(* PLC project Untitled1, Eindhoven University of Technology (TU/e) CIF to Structured Text 0.0 *)
(* stored: creationDateTime 1970-01-01T01:00:00 *)

TYPE STATE : STRUCT
  curTime : LREAL;
  dvar_M_BoolToEventsDH AT %Q* : enum_E;
  dvar_M_BoolToEventsP AT %Q* : enum_E;
  dvar_M_BoolToEventsS AT %Q* : enum_E;
  dvar_M_BoolToEventsTB AT %Q* : enum_E;
  cvar_M_BTimer1_t AT %Q* : LREAL;
  dvar_M_BTimer1 AT %Q* : enum_E;
  dvar_M_HardwareMapDH_out_a_Dstartled AT %Q* : BOOL;
  dvar_M_HardwareMapDH_out_a_Dresetled AT %Q* : BOOL;
  dvar_M_HardwareMapDH_out_a_DledQ1 AT %Q* : BOOL;
  dvar_M_HardwareMapDH_out_a_DledQ2 AT %Q* : BOOL;
  dvar_M_HardwareMapDH_out_a_Dout4 AT %Q* : BOOL;
  dvar_M_HardwareMapDH_out_a_Dout5 AT %Q* : BOOL;
  dvar_M_HardwareMapDH_out_a_Dout6 AT %Q* : BOOL;
  dvar_M_HardwareMapDH_out_a_Dout7 AT %Q* : BOOL;
  dvar_M_HardwareMapDH_out_a_pusher1 AT %Q* : BOOL;
  dvar_M_HardwareMapDH_out_a_pusher2 AT %Q* : BOOL;
  dvar_M_HardwareMapDH_out_a_pusher3 AT %Q* : BOOL;
  dvar_M_HardwareMapDH_out_a_Hstartled AT %Q* : BOOL;
  dvar_M_HardwareMapDH_out_a_Hresetled AT %Q* : BOOL;
  dvar_M_HardwareMapDH_out_a_HledQ1 AT %Q* : BOOL;
  dvar_M_HardwareMapDH_out_a_HledQ2 AT %Q* : BOOL;
  dvar_M_HardwareMapDH_out_a_Hout4 AT %Q* : BOOL;
  dvar_M_HardwareMapDH_out_a_Hout5 AT %Q* : BOOL;
  dvar_M_HardwareMapDH_out_a_Hout6 AT %Q* : BOOL;
  dvar_M_HardwareMapDH_out_a_Hout7 AT %Q* : BOOL;
  dvar_M_HardwareMapDH_out_a_x2distributing AT %Q* : BOOL;
  dvar_M_HardwareMapDH_out_a_x2testing AT %Q* : BOOL;
  dvar_M_HardwareMapDH_out_a_zdown AT %Q* : BOOL;
  dvar_M_HardwareMapDH_out_a_gripperclose AT %Q* : BOOL;
  dvar_M_HardwareMapDH_out_a_transfer2pickpos AT %Q* : BOOL;
  dvar_M_HardwareMapDH_out_a_transfer2droppos AT %Q* : BOOL;
  dvar_M_HardwareMapDH_out_a_vacuum AT %Q* : BOOL;
  dvar_M_HardwareMapDH_out_a_ejectpulse AT %Q* : BOOL;
  dvar_M_HardwareMapDH_out_a_handlingready AT %Q* : BOOL;
  dvar_M_HardwareMapDH_init_err_sen_idx AT %Q* : DINT;
  dvar_M_HardwareMapDH_init_err_led_idx AT %Q* : DINT;
  cvar_M_HardwareMapDH_t AT %Q* : LREAL;
  dvar_M_HardwareMapDH AT %Q* : enum_E;
  dvar_M_HardwareMapP_out_a_Pstartled AT %Q* : BOOL;
  dvar_M_HardwareMapP_out_a_Presetled AT %Q* : BOOL;
  dvar_M_HardwareMapP_out_a_PledQ1 AT %Q* : BOOL;
  dvar_M_HardwareMapP_out_a_PledQ2 AT %Q* : BOOL;
  dvar_M_HardwareMapP_out_a_Pout4 AT %Q* : BOOL;
  dvar_M_HardwareMapP_out_a_Pout5 AT %Q* : BOOL;
  dvar_M_HardwareMapP_out_a_Pout6 AT %Q* : BOOL;
  dvar_M_HardwareMapP_out_a_Pout7 AT %Q* : BOOL;
  dvar_M_HardwareMapP_out_a_drill AT %Q* : BOOL;
  dvar_M_HardwareMapP_out_a_turntable AT %Q* : BOOL;
  dvar_M_HardwareMapP_out_a_drilldown AT %Q* : BOOL;
  dvar_M_HardwareMapP_out_a_drillup AT %Q* : BOOL;
  dvar_M_HardwareMapP_out_a_clamp AT %Q* : BOOL;
  dvar_M_HardwareMapP_out_a_tester AT %Q* : BOOL;
  dvar_M_HardwareMapP_out_a_eject AT %Q* : BOOL;
  dvar_M_HardwareMapP_out_a_processingready AT %Q* : BOOL;
  dvar_M_HardwareMapP_init_err_sen_idx AT %Q* : DINT;
  dvar_M_HardwareMapP_init_err_led_idx AT %Q* : DINT;
  cvar_M_HardwareMapP_t AT %Q* : LREAL;
  dvar_M_HardwareMapP AT %Q* : enum_E;
  dvar_M_HardwareMapS_out_a_Sstartled AT %Q* : BOOL;
  dvar_M_HardwareMapS_out_a_Sresetled AT %Q* : BOOL;
  dvar_M_HardwareMapS_out_a_SledQ1 AT %Q* : BOOL;
  dvar_M_HardwareMapS_out_a_SledQ2 AT %Q* : BOOL;
  dvar_M_HardwareMapS_out_a_Sout4 AT %Q* : BOOL;
  dvar_M_HardwareMapS_out_a_Sout5 AT %Q* : BOOL;
  dvar_M_HardwareMapS_out_a_Sout6 AT %Q* : BOOL;
  dvar_M_HardwareMapS_out_a_Sout7 AT %Q* : BOOL;
  dvar_M_HardwareMapS_out_a_conveyer AT %Q* : BOOL;
  dvar_M_HardwareMapS_out_a_gate1 AT %Q* : BOOL;
  dvar_M_HardwareMapS_out_a_gate2 AT %Q* : BOOL;
  dvar_M_HardwareMapS_out_a_stopperretract AT %Q* : BOOL;
  dvar_M_HardwareMapS_out_a_sortingready AT %Q* : BOOL;
  dvar_M_HardwareMapS_init_err_sen_idx AT %Q* : DINT;
  dvar_M_HardwareMapS_init_err_led_idx AT %Q* : DINT;
  cvar_M_HardwareMapS_t AT %Q* : LREAL;
  dvar_M_HardwareMapS AT %Q* : enum_E;
  dvar_M_HardwareMapTB_out_a_Tstartled AT %Q* : BOOL;
  dvar_M_HardwareMapTB_out_a_Tresetled AT %Q* : BOOL;
  dvar_M_HardwareMapTB_out_a_TledQ1 AT %Q* : BOOL;
  dvar_M_HardwareMapTB_out_a_TledQ2 AT %Q* : BOOL;
  dvar_M_HardwareMapTB_out_a_Tout4 AT %Q* : BOOL;
  dvar_M_HardwareMapTB_out_a_Tout5 AT %Q* : BOOL;
  dvar_M_HardwareMapTB_out_a_Tout6 AT %Q* : BOOL;
  dvar_M_HardwareMapTB_out_a_Tout7 AT %Q* : BOOL;
  dvar_M_HardwareMapTB_out_a_elevator_up AT %Q* : BOOL;
  dvar_M_HardwareMapTB_out_a_elevator_down AT %Q* : BOOL;
  dvar_M_HardwareMapTB_out_a_pusher AT %Q* : BOOL;
  dvar_M_HardwareMapTB_out_a_airslide AT %Q* : BOOL;
  dvar_M_HardwareMapTB_out_a_testingready AT %Q* : BOOL;
  dvar_M_HardwareMapTB_out_a_Bstartled AT %Q* : BOOL;
  dvar_M_HardwareMapTB_out_a_Bresetled AT %Q* : BOOL;
  dvar_M_HardwareMapTB_out_a_BledQ1 AT %Q* : BOOL;
  dvar_M_HardwareMapTB_out_a_BledQ2 AT %Q* : BOOL;
  dvar_M_HardwareMapTB_out_a_Bout4 AT %Q* : BOOL;
  dvar_M_HardwareMapTB_out_a_Bout5 AT %Q* : BOOL;
  dvar_M_HardwareMapTB_out_a_Bout6 AT %Q* : BOOL;
  dvar_M_HardwareMapTB_out_a_Bout7 AT %Q* : BOOL;
  dvar_M_HardwareMapTB_out_a_separator AT %Q* : BOOL;
  dvar_M_HardwareMapTB_out_a_conveyerB AT %Q* : BOOL;
  dvar_M_HardwareMapTB_out_a_bufferingready AT %Q* : BOOL;
  dvar_M_HardwareMapTB_init_err_sen_idx AT %Q* : DINT;
  dvar_M_HardwareMapTB_init_err_led_idx AT %Q* : DINT;
  cvar_M_HardwareMapTB_t AT %Q* : LREAL;
  dvar_M_HardwareMapTB AT %Q* : enum_E;
  cvar_M_STimer1_t AT %Q* : LREAL;
  dvar_M_STimer1 AT %Q* : enum_E;
  dvar_M_sup_A_airslide AT %Q* : enum_E;
  dvar_M_sup_A_bufferingready AT %Q* : enum_E;
  dvar_M_sup_A_clamp AT %Q* : enum_E;
  dvar_M_sup_A_conveyer AT %Q* : enum_E;
  dvar_M_sup_A_conveyerB AT %Q* : enum_E;
  dvar_M_sup_A_drill AT %Q* : enum_E;
  dvar_M_sup_A_drilldown AT %Q* : enum_E;
  dvar_M_sup_A_drillup AT %Q* : enum_E;
  dvar_M_sup_A_eject AT %Q* : enum_E;
  dvar_M_sup_A_ejectpulse AT %Q* : enum_E;
  dvar_M_sup_A_elevator_down AT %Q* : enum_E;
  dvar_M_sup_A_elevator_up AT %Q* : enum_E;
  dvar_M_sup_A_gate1 AT %Q* : enum_E;
  dvar_M_sup_A_gate2 AT %Q* : enum_E;
  dvar_M_sup_A_gripperclose AT %Q* : enum_E;
  dvar_M_sup_A_handlingready AT %Q* : enum_E;
  dvar_M_sup_A_processingready AT %Q* : enum_E;
  dvar_M_sup_A_pusher AT %Q* : enum_E;
  dvar_M_sup_A_pusher1 AT %Q* : enum_E;
  dvar_M_sup_A_pusher2 AT %Q* : enum_E;
  dvar_M_sup_A_pusher3 AT %Q* : enum_E;
  dvar_M_sup_A_separator AT %Q* : enum_E;
  dvar_M_sup_A_sortingready AT %Q* : enum_E;
  dvar_M_sup_A_stopperretract AT %Q* : enum_E;
  dvar_M_sup_A_tester AT %Q* : enum_E;
  dvar_M_sup_A_testingready AT %Q* : enum_E;
  dvar_M_sup_A_transfer2droppos AT %Q* : enum_E;
  dvar_M_sup_A_transfer2pickpos AT %Q* : enum_E;
  dvar_M_sup_A_turntable AT %Q* : enum_E;
  dvar_M_sup_A_vacuum AT %Q* : enum_E;
  dvar_M_sup_A_x2distributing AT %Q* : enum_E;
  dvar_M_sup_A_x2testing AT %Q* : enum_E;
  dvar_M_sup_A_zdown AT %Q* : enum_E;
  dvar_M_sup_BDynamics AT %Q* : enum_E;
  dvar_M_sup_BTimer AT %Q* : enum_E;
  dvar_M_sup_ClampDrill AT %Q* : enum_E;
  dvar_M_sup_DDynamics1 AT %Q* : enum_E;
  dvar_M_sup_DDynamics2 AT %Q* : enum_E;
  dvar_M_sup_DDynamics3 AT %Q* : enum_E;
  dvar_M_sup_HDynamics1 AT %Q* : enum_E;
  dvar_M_sup_HDynamics2 AT %Q* : enum_E;
  dvar_M_sup_HDynamics3 AT %Q* : enum_E;
  dvar_M_sup_PDynamics AT %Q* : enum_E;
  dvar_M_sup_PusherLift AT %Q* : enum_E;
  dvar_M_sup_S_atdrill AT %Q* : enum_E;
  dvar_M_sup_S_atend AT %Q* : enum_E;
  dvar_M_sup_S_atexit AT %Q* : enum_E;
  dvar_M_sup_S_atin AT %Q* : enum_E;
  dvar_M_sup_S_atinput AT %Q* : enum_E;
  dvar_M_sup_S_atseparator AT %Q* : enum_E;
  dvar_M_sup_S_atspare AT %Q* : enum_E;
  dvar_M_sup_S_attest AT %Q* : enum_E;
  dvar_M_sup_S_Binitialized AT %Q* : enum_E;
  dvar_M_sup_S_bufferingbusy AT %Q* : enum_E;
  dvar_M_sup_S_capacitive AT %Q* : enum_E;
  dvar_M_sup_S_clamp AT %Q* : enum_E;
  dvar_M_sup_S_Dinitialized AT %Q* : enum_E;
  dvar_M_sup_S_drill_down AT %Q* : enum_E;
  dvar_M_sup_S_drill_up AT %Q* : enum_E;
  dvar_M_sup_S_elevator_down AT %Q* : enum_E;
  dvar_M_sup_S_elevator_up AT %Q* : enum_E;
  dvar_M_sup_S_gate1_closed AT %Q* : enum_E;
  dvar_M_sup_S_gate1_opened AT %Q* : enum_E;
  dvar_M_sup_S_gate2_closed AT %Q* : enum_E;
  dvar_M_sup_S_gate2_opened AT %Q* : enum_E;
  dvar_M_sup_S_gripper AT %Q* : enum_E;
  dvar_M_sup_S_handlingbusy AT %Q* : enum_E;
  dvar_M_sup_S_Hinitialized AT %Q* : enum_E;
  dvar_M_sup_S_inductive AT %Q* : enum_E;
  dvar_M_sup_S_optical AT %Q* : enum_E;
  dvar_M_sup_S_opticalT AT %Q* : enum_E;
  dvar_M_sup_S_Pinitialized AT %Q* : enum_E;
  dvar_M_sup_S_processingbusy AT %Q* : enum_E;
  dvar_M_sup_S_product AT %Q* : enum_E;
  dvar_M_sup_S_product1 AT %Q* : enum_E;
  dvar_M_sup_S_product2 AT %Q* : enum_E;
  dvar_M_sup_S_product3 AT %Q* : enum_E;
  dvar_M_sup_S_product4 AT %Q* : enum_E;
  dvar_M_sup_S_productheight AT %Q* : enum_E;
  dvar_M_sup_S_pusher AT %Q* : enum_E;
  dvar_M_sup_S_pusher1_in AT %Q* : enum_E;
  dvar_M_sup_S_pusher1_out AT %Q* : enum_E;
  dvar_M_sup_S_pusher2_in AT %Q* : enum_E;
  dvar_M_sup_S_pusher2_out AT %Q* : enum_E;
  dvar_M_sup_S_pusher3_in AT %Q* : enum_E;
  dvar_M_sup_S_pusher3_out AT %Q* : enum_E;
  dvar_M_sup_S_reflective AT %Q* : enum_E;
  dvar_M_sup_S_separator_closed AT %Q* : enum_E;
  dvar_M_sup_S_separator_opened AT %Q* : enum_E;
  dvar_M_sup_S_Sinitialized AT %Q* : enum_E;
  dvar_M_sup_S_slidefull AT %Q* : enum_E;
  dvar_M_sup_S_sortingbusy AT %Q* : enum_E;
  dvar_M_sup_S_stack1_filled AT %Q* : enum_E;
  dvar_M_sup_S_stack2_filled AT %Q* : enum_E;
  dvar_M_sup_S_stack3_filled AT %Q* : enum_E;
  dvar_M_sup_S_test_ok AT %Q* : enum_E;
  dvar_M_sup_S_testingbusy AT %Q* : enum_E;
  dvar_M_sup_S_Tinitialized AT %Q* : enum_E;
  dvar_M_sup_S_transfer_atdrop AT %Q* : enum_E;
  dvar_M_sup_S_transfer_athalfway AT %Q* : enum_E;
  dvar_M_sup_S_transfer_atpickup AT %Q* : enum_E;
  dvar_M_sup_S_turntable AT %Q* : enum_E;
  dvar_M_sup_S_vacuum AT %Q* : enum_E;
  dvar_M_sup_S_xpos_at1 AT %Q* : enum_E;
  dvar_M_sup_S_xpos_at2 AT %Q* : enum_E;
  dvar_M_sup_S_xpos_at3 AT %Q* : enum_E;
  dvar_M_sup_S_xpos_atdrop AT %Q* : enum_E;
  dvar_M_sup_S_zpos_atdown AT %Q* : enum_E;
  dvar_M_sup_S_zpos_atup AT %Q* : enum_E;
  dvar_M_sup_SDynamics1 AT %Q* : enum_E;
  dvar_M_sup_SDynamics2 AT %Q* : enum_E;
  dvar_M_sup_STimer AT %Q* : enum_E;
  dvar_M_sup_sup AT %Q* : enum_E;
  dvar_M_sup_TDynamics AT %Q* : enum_E;
  dvar_M_sup_Tester AT %Q* : enum_E;
  dvar_M_sup_Timer AT %Q* : enum_E;
  dvar_M_sup_TTimer AT %Q* : enum_E;
  cvar_M_Timer1_t AT %Q* : LREAL;
  dvar_M_Timer1 AT %Q* : enum_E;
  cvar_M_TTimer1_t AT %Q* : LREAL;
  dvar_M_TTimer1 AT %Q* : enum_E;
END_STRUCT;
END_TYPE

TYPE enum_E : (elit_eight, elit_five, elit_Four, elit_four2, elit_init0, elit_init1, elit_init2, elit_init3, elit_init4, elit_init5, elit_init6, elit_init7, elit_init8, elit_init9, elit_init_error, elit_init_ok, elit_init_sensor_check, elit_initialized, elit_nine, elit_Off, elit_On, elit_One, elit_one2, elit_Running, elit_seven, elit_six, elit_Three, elit_three2, elit_Timeout, elit_Two, elit_two2, elit_X);
END_TYPE

FUNCTION ifExprFunc1 : LREAL
  VAR_INPUT
    state : STATE;
  END_VAR

            IF ((state.dvar_M_BTimer1) = (elit_Running)) THEN
    ifExprFunc1 := 1.0;
ELSE
    ifExprFunc1 := 0.0;
END_IF;
          
END_FUNCTION

FUNCTION derivcvar_M_BTimer1_t : LREAL
  VAR_INPUT
    state : STATE;
  END_VAR

            derivcvar_M_BTimer1_t := ifExprFunc1(state);
          
END_FUNCTION

FUNCTION derivcvar_M_HardwareMapDH_t : LREAL
  VAR_INPUT
    state : STATE;
  END_VAR

            derivcvar_M_HardwareMapDH_t := 1.0;
          
END_FUNCTION

FUNCTION derivcvar_M_HardwareMapP_t : LREAL
  VAR_INPUT
    state : STATE;
  END_VAR

            derivcvar_M_HardwareMapP_t := 1.0;
          
END_FUNCTION

FUNCTION derivcvar_M_HardwareMapS_t : LREAL
  VAR_INPUT
    state : STATE;
  END_VAR

            derivcvar_M_HardwareMapS_t := 1.0;
          
END_FUNCTION

FUNCTION derivcvar_M_HardwareMapTB_t : LREAL
  VAR_INPUT
    state : STATE;
  END_VAR

            derivcvar_M_HardwareMapTB_t := 1.0;
          
END_FUNCTION

FUNCTION ifExprFunc2 : LREAL
  VAR_INPUT
    state : STATE;
  END_VAR

            IF ((state.dvar_M_STimer1) = (elit_Running)) THEN
    ifExprFunc2 := 1.0;
ELSE
    ifExprFunc2 := 0.0;
END_IF;
          
END_FUNCTION

FUNCTION derivcvar_M_STimer1_t : LREAL
  VAR_INPUT
    state : STATE;
  END_VAR

            derivcvar_M_STimer1_t := ifExprFunc2(state);
          
END_FUNCTION

FUNCTION ifExprFunc3 : LREAL
  VAR_INPUT
    state : STATE;
  END_VAR

            IF ((state.dvar_M_Timer1) = (elit_Running)) THEN
    ifExprFunc3 := 1.0;
ELSE
    ifExprFunc3 := 0.0;
END_IF;
          
END_FUNCTION

FUNCTION derivcvar_M_Timer1_t : LREAL
  VAR_INPUT
    state : STATE;
  END_VAR

            derivcvar_M_Timer1_t := ifExprFunc3(state);
          
END_FUNCTION

FUNCTION ifExprFunc4 : LREAL
  VAR_INPUT
    state : STATE;
  END_VAR

            IF ((state.dvar_M_TTimer1) = (elit_Running)) THEN
    ifExprFunc4 := 1.0;
ELSE
    ifExprFunc4 := 0.0;
END_IF;
          
END_FUNCTION

FUNCTION derivcvar_M_TTimer1_t : LREAL
  VAR_INPUT
    state : STATE;
  END_VAR

            derivcvar_M_TTimer1_t := ifExprFunc4(state);
          
END_FUNCTION

PROGRAM MAIN
  VAR_OUTPUT
    timerValue0 : TIME;
    timerValue1 : TIME;
  END_VAR
  VAR
    cnt : LINT;
    first : BOOL := TRUE;
    curTimerValue : TIME;
    state0 : STATE;
    curTime : LREAL;
    loopsKilled : LINT;
  END_VAR
  VAR_TEMP
    lastTimerValue : TIME;
    curDeltaTime : TIME;
    curDeltaSecs : LREAL;
    state1 : STATE;
    progress : BOOL;
    loopCount : INT;
    b1 : BOOL;
    b2 : BOOL;
    b3 : BOOL;
    b4 : BOOL;
  END_VAR

            
// Handle 'time' and cycle time.
cnt := cnt + 1;

timer0(IN := curTimer = 0, PT := T#1D);
timer1(IN := curTimer = 1, PT := T#1D);
timerValue0 := timer0.ET;
timerValue1 := timer1.ET;

lastTimerValue := curTimerValue;
IF curTimer = 0 THEN
    curTimerValue := timerValue0;
ELSE
    curTimerValue := timerValue1;
END_IF;
curDeltaTime := curTimerValue - lastTimerValue;
curDeltaSecs := TIME_TO_LREAL(curDeltaTime) / 1000;
curTime := curTime + curDeltaSecs;

IF cnt MOD 10 = 0 THEN
    curTimer := 1 - curTimer;
    curTimerValue := T#0S;
    timer0(IN := curTimer = 0, PT := T#1D);
    timer1(IN := curTimer = 1, PT := T#1D);
    timerValue0 := timer0.ET;
    timerValue1 := timer1.ET;
END_IF;

IF first THEN
    first := FALSE;

    // Initialize state variables for initial state.
    state0.dvar_M_BoolToEventsDH := elit_X;
    state0.dvar_M_BoolToEventsP := elit_X;
    state0.dvar_M_BoolToEventsS := elit_X;
    state0.dvar_M_BoolToEventsTB := elit_X;
    state0.cvar_M_BTimer1_t := 0.0;
    state0.dvar_M_BTimer1 := elit_Off;
    state0.dvar_M_HardwareMapDH_out_a_Dstartled := FALSE;
    state0.dvar_M_HardwareMapDH_out_a_Dresetled := FALSE;
    state0.dvar_M_HardwareMapDH_out_a_DledQ1 := TRUE;
    state0.dvar_M_HardwareMapDH_out_a_DledQ2 := TRUE;
    state0.dvar_M_HardwareMapDH_out_a_Dout4 := FALSE;
    state0.dvar_M_HardwareMapDH_out_a_Dout5 := FALSE;
    state0.dvar_M_HardwareMapDH_out_a_Dout6 := FALSE;
    state0.dvar_M_HardwareMapDH_out_a_Dout7 := FALSE;
    state0.dvar_M_HardwareMapDH_out_a_pusher1 := FALSE;
    state0.dvar_M_HardwareMapDH_out_a_pusher2 := FALSE;
    state0.dvar_M_HardwareMapDH_out_a_pusher3 := FALSE;
    state0.dvar_M_HardwareMapDH_out_a_Hstartled := FALSE;
    state0.dvar_M_HardwareMapDH_out_a_Hresetled := FALSE;
    state0.dvar_M_HardwareMapDH_out_a_HledQ1 := TRUE;
    state0.dvar_M_HardwareMapDH_out_a_HledQ2 := TRUE;
    state0.dvar_M_HardwareMapDH_out_a_Hout4 := FALSE;
    state0.dvar_M_HardwareMapDH_out_a_Hout5 := FALSE;
    state0.dvar_M_HardwareMapDH_out_a_Hout6 := FALSE;
    state0.dvar_M_HardwareMapDH_out_a_Hout7 := FALSE;
    state0.dvar_M_HardwareMapDH_out_a_x2distributing := TRUE;
    state0.dvar_M_HardwareMapDH_out_a_x2testing := TRUE;
    state0.dvar_M_HardwareMapDH_out_a_zdown := FALSE;
    state0.dvar_M_HardwareMapDH_out_a_gripperclose := FALSE;
    state0.dvar_M_HardwareMapDH_out_a_transfer2pickpos := FALSE;
    state0.dvar_M_HardwareMapDH_out_a_transfer2droppos := FALSE;
    state0.dvar_M_HardwareMapDH_out_a_vacuum := FALSE;
    state0.dvar_M_HardwareMapDH_out_a_ejectpulse := FALSE;
    state0.dvar_M_HardwareMapDH_out_a_handlingready := FALSE;
    state0.dvar_M_HardwareMapDH_init_err_sen_idx := -1;
    state0.dvar_M_HardwareMapDH_init_err_led_idx := 0;
    state0.cvar_M_HardwareMapDH_t := 0.0;
    state0.dvar_M_HardwareMapDH := elit_init0;
    state0.dvar_M_HardwareMapP_out_a_Pstartled := FALSE;
    state0.dvar_M_HardwareMapP_out_a_Presetled := FALSE;
    state0.dvar_M_HardwareMapP_out_a_PledQ1 := TRUE;
    state0.dvar_M_HardwareMapP_out_a_PledQ2 := TRUE;
    state0.dvar_M_HardwareMapP_out_a_Pout4 := FALSE;
    state0.dvar_M_HardwareMapP_out_a_Pout5 := FALSE;
    state0.dvar_M_HardwareMapP_out_a_Pout6 := FALSE;
    state0.dvar_M_HardwareMapP_out_a_Pout7 := FALSE;
    state0.dvar_M_HardwareMapP_out_a_drill := FALSE;
    state0.dvar_M_HardwareMapP_out_a_turntable := FALSE;
    state0.dvar_M_HardwareMapP_out_a_drilldown := FALSE;
    state0.dvar_M_HardwareMapP_out_a_drillup := TRUE;
    state0.dvar_M_HardwareMapP_out_a_clamp := FALSE;
    state0.dvar_M_HardwareMapP_out_a_tester := FALSE;
    state0.dvar_M_HardwareMapP_out_a_eject := FALSE;
    state0.dvar_M_HardwareMapP_out_a_processingready := FALSE;
    state0.dvar_M_HardwareMapP_init_err_sen_idx := -1;
    state0.dvar_M_HardwareMapP_init_err_led_idx := 0;
    state0.cvar_M_HardwareMapP_t := 0.0;
    state0.dvar_M_HardwareMapP := elit_init0;
    state0.dvar_M_HardwareMapS_out_a_Sstartled := FALSE;
    state0.dvar_M_HardwareMapS_out_a_Sresetled := FALSE;
    state0.dvar_M_HardwareMapS_out_a_SledQ1 := TRUE;
    state0.dvar_M_HardwareMapS_out_a_SledQ2 := TRUE;
    state0.dvar_M_HardwareMapS_out_a_Sout4 := FALSE;
    state0.dvar_M_HardwareMapS_out_a_Sout5 := FALSE;
    state0.dvar_M_HardwareMapS_out_a_Sout6 := FALSE;
    state0.dvar_M_HardwareMapS_out_a_Sout7 := FALSE;
    state0.dvar_M_HardwareMapS_out_a_conveyer := FALSE;
    state0.dvar_M_HardwareMapS_out_a_gate1 := FALSE;
    state0.dvar_M_HardwareMapS_out_a_gate2 := FALSE;
    state0.dvar_M_HardwareMapS_out_a_stopperretract := FALSE;
    state0.dvar_M_HardwareMapS_out_a_sortingready := FALSE;
    state0.dvar_M_HardwareMapS_init_err_sen_idx := -1;
    state0.dvar_M_HardwareMapS_init_err_led_idx := 0;
    state0.cvar_M_HardwareMapS_t := 0.0;
    state0.dvar_M_HardwareMapS := elit_init0;
    state0.dvar_M_HardwareMapTB_out_a_Tstartled := FALSE;
    state0.dvar_M_HardwareMapTB_out_a_Tresetled := FALSE;
    state0.dvar_M_HardwareMapTB_out_a_TledQ1 := TRUE;
    state0.dvar_M_HardwareMapTB_out_a_TledQ2 := TRUE;
    state0.dvar_M_HardwareMapTB_out_a_Tout4 := FALSE;
    state0.dvar_M_HardwareMapTB_out_a_Tout5 := FALSE;
    state0.dvar_M_HardwareMapTB_out_a_Tout6 := FALSE;
    state0.dvar_M_HardwareMapTB_out_a_Tout7 := FALSE;
    state0.dvar_M_HardwareMapTB_out_a_elevator_up := FALSE;
    state0.dvar_M_HardwareMapTB_out_a_elevator_down := TRUE;
    state0.dvar_M_HardwareMapTB_out_a_pusher := FALSE;
    state0.dvar_M_HardwareMapTB_out_a_airslide := FALSE;
    state0.dvar_M_HardwareMapTB_out_a_testingready := FALSE;
    state0.dvar_M_HardwareMapTB_out_a_Bstartled := FALSE;
    state0.dvar_M_HardwareMapTB_out_a_Bresetled := FALSE;
    state0.dvar_M_HardwareMapTB_out_a_BledQ1 := TRUE;
    state0.dvar_M_HardwareMapTB_out_a_BledQ2 := TRUE;
    state0.dvar_M_HardwareMapTB_out_a_Bout4 := FALSE;
    state0.dvar_M_HardwareMapTB_out_a_Bout5 := FALSE;
    state0.dvar_M_HardwareMapTB_out_a_Bout6 := FALSE;
    state0.dvar_M_HardwareMapTB_out_a_Bout7 := FALSE;
    state0.dvar_M_HardwareMapTB_out_a_separator := FALSE;
    state0.dvar_M_HardwareMapTB_out_a_conveyerB := FALSE;
    state0.dvar_M_HardwareMapTB_out_a_bufferingready := FALSE;
    state0.dvar_M_HardwareMapTB_init_err_sen_idx := -1;
    state0.dvar_M_HardwareMapTB_init_err_led_idx := 0;
    state0.cvar_M_HardwareMapTB_t := 0.0;
    state0.dvar_M_HardwareMapTB := elit_init0;
    state0.cvar_M_STimer1_t := 0.0;
    state0.dvar_M_STimer1 := elit_Off;
    state0.dvar_M_sup_A_airslide := elit_Off;
    state0.dvar_M_sup_A_bufferingready := elit_Off;
    state0.dvar_M_sup_A_clamp := elit_Off;
    state0.dvar_M_sup_A_conveyer := elit_Off;
    state0.dvar_M_sup_A_conveyerB := elit_Off;
    state0.dvar_M_sup_A_drill := elit_Off;
    state0.dvar_M_sup_A_drilldown := elit_Off;
    state0.dvar_M_sup_A_drillup := elit_On;
    state0.dvar_M_sup_A_eject := elit_Off;
    state0.dvar_M_sup_A_ejectpulse := elit_Off;
    state0.dvar_M_sup_A_elevator_down := elit_On;
    state0.dvar_M_sup_A_elevator_up := elit_Off;
    state0.dvar_M_sup_A_gate1 := elit_Off;
    state0.dvar_M_sup_A_gate2 := elit_Off;
    state0.dvar_M_sup_A_gripperclose := elit_Off;
    state0.dvar_M_sup_A_handlingready := elit_Off;
    state0.dvar_M_sup_A_processingready := elit_Off;
    state0.dvar_M_sup_A_pusher := elit_Off;
    state0.dvar_M_sup_A_pusher1 := elit_Off;
    state0.dvar_M_sup_A_pusher2 := elit_Off;
    state0.dvar_M_sup_A_pusher3 := elit_Off;
    state0.dvar_M_sup_A_separator := elit_On;
    state0.dvar_M_sup_A_sortingready := elit_Off;
    state0.dvar_M_sup_A_stopperretract := elit_Off;
    state0.dvar_M_sup_A_tester := elit_Off;
    state0.dvar_M_sup_A_testingready := elit_Off;
    state0.dvar_M_sup_A_transfer2droppos := elit_Off;
    state0.dvar_M_sup_A_transfer2pickpos := elit_Off;
    state0.dvar_M_sup_A_turntable := elit_Off;
    state0.dvar_M_sup_A_vacuum := elit_Off;
    state0.dvar_M_sup_A_x2distributing := elit_On;
    state0.dvar_M_sup_A_x2testing := elit_On;
    state0.dvar_M_sup_A_zdown := elit_Off;
    state0.dvar_M_sup_BDynamics := elit_X;
    state0.dvar_M_sup_BTimer := elit_Off;
    state0.dvar_M_sup_ClampDrill := elit_one2;
    state0.dvar_M_sup_DDynamics1 := elit_X;
    state0.dvar_M_sup_DDynamics2 := elit_X;
    state0.dvar_M_sup_DDynamics3 := elit_X;
    state0.dvar_M_sup_HDynamics1 := elit_X;
    state0.dvar_M_sup_HDynamics2 := elit_X;
    state0.dvar_M_sup_HDynamics3 := elit_X;
    state0.dvar_M_sup_PDynamics := elit_X;
    state0.dvar_M_sup_PusherLift := elit_One;
    state0.dvar_M_sup_S_atdrill := elit_Off;
    state0.dvar_M_sup_S_atend := elit_Off;
    state0.dvar_M_sup_S_atexit := elit_Off;
    state0.dvar_M_sup_S_atin := elit_Off;
    state0.dvar_M_sup_S_atinput := elit_Off;
    state0.dvar_M_sup_S_atseparator := elit_Off;
    state0.dvar_M_sup_S_atspare := elit_Off;
    state0.dvar_M_sup_S_attest := elit_Off;
    state0.dvar_M_sup_S_Binitialized := elit_Off;
    state0.dvar_M_sup_S_bufferingbusy := elit_On;
    state0.dvar_M_sup_S_capacitive := elit_Off;
    state0.dvar_M_sup_S_clamp := elit_Off;
    state0.dvar_M_sup_S_Dinitialized := elit_Off;
    state0.dvar_M_sup_S_drill_down := elit_Off;
    state0.dvar_M_sup_S_drill_up := elit_On;
    state0.dvar_M_sup_S_elevator_down := elit_On;
    state0.dvar_M_sup_S_elevator_up := elit_Off;
    state0.dvar_M_sup_S_gate1_closed := elit_Off;
    state0.dvar_M_sup_S_gate1_opened := elit_On;
    state0.dvar_M_sup_S_gate2_closed := elit_Off;
    state0.dvar_M_sup_S_gate2_opened := elit_On;
    state0.dvar_M_sup_S_gripper := elit_Off;
    state0.dvar_M_sup_S_handlingbusy := elit_On;
    state0.dvar_M_sup_S_Hinitialized := elit_Off;
    state0.dvar_M_sup_S_inductive := elit_Off;
    state0.dvar_M_sup_S_optical := elit_Off;
    state0.dvar_M_sup_S_opticalT := elit_Off;
    state0.dvar_M_sup_S_Pinitialized := elit_Off;
    state0.dvar_M_sup_S_processingbusy := elit_On;
    state0.dvar_M_sup_S_product := elit_Off;
    state0.dvar_M_sup_S_product1 := elit_Off;
    state0.dvar_M_sup_S_product2 := elit_Off;
    state0.dvar_M_sup_S_product3 := elit_Off;
    state0.dvar_M_sup_S_product4 := elit_Off;
    state0.dvar_M_sup_S_productheight := elit_Off;
    state0.dvar_M_sup_S_pusher := elit_Off;
    state0.dvar_M_sup_S_pusher1_in := elit_On;
    state0.dvar_M_sup_S_pusher1_out := elit_Off;
    state0.dvar_M_sup_S_pusher2_in := elit_On;
    state0.dvar_M_sup_S_pusher2_out := elit_Off;
    state0.dvar_M_sup_S_pusher3_in := elit_On;
    state0.dvar_M_sup_S_pusher3_out := elit_Off;
    state0.dvar_M_sup_S_reflective := elit_Off;
    state0.dvar_M_sup_S_separator_closed := elit_On;
    state0.dvar_M_sup_S_separator_opened := elit_Off;
    state0.dvar_M_sup_S_Sinitialized := elit_Off;
    state0.dvar_M_sup_S_slidefull := elit_Off;
    state0.dvar_M_sup_S_sortingbusy := elit_On;
    state0.dvar_M_sup_S_stack1_filled := elit_On;
    state0.dvar_M_sup_S_stack2_filled := elit_On;
    state0.dvar_M_sup_S_stack3_filled := elit_On;
    state0.dvar_M_sup_S_test_ok := elit_Off;
    state0.dvar_M_sup_S_testingbusy := elit_On;
    state0.dvar_M_sup_S_Tinitialized := elit_Off;
    state0.dvar_M_sup_S_transfer_atdrop := elit_Off;
    state0.dvar_M_sup_S_transfer_athalfway := elit_On;
    state0.dvar_M_sup_S_transfer_atpickup := elit_Off;
    state0.dvar_M_sup_S_turntable := elit_On;
    state0.dvar_M_sup_S_vacuum := elit_Off;
    state0.dvar_M_sup_S_xpos_at1 := elit_Off;
    state0.dvar_M_sup_S_xpos_at2 := elit_Off;
    state0.dvar_M_sup_S_xpos_at3 := elit_Off;
    state0.dvar_M_sup_S_xpos_atdrop := elit_On;
    state0.dvar_M_sup_S_zpos_atdown := elit_Off;
    state0.dvar_M_sup_S_zpos_atup := elit_On;
    state0.dvar_M_sup_SDynamics1 := elit_X;
    state0.dvar_M_sup_SDynamics2 := elit_X;
    state0.dvar_M_sup_STimer := elit_Off;
    state0.dvar_M_sup_sup := elit_X;
    state0.dvar_M_sup_TDynamics := elit_X;
    state0.dvar_M_sup_Tester := elit_One;
    state0.dvar_M_sup_Timer := elit_Off;
    state0.dvar_M_sup_TTimer := elit_Off;
    state0.cvar_M_Timer1_t := 0.0;
    state0.dvar_M_Timer1 := elit_Off;
    state0.cvar_M_TTimer1_t := 0.0;
    state0.dvar_M_TTimer1 := elit_Off;
ELSE
    // Update continuous variables for time delay.
    state1.cvar_M_BTimer1_t := state0.cvar_M_BTimer1_t + curDeltaSecs * derivcvar_M_BTimer1_t(state0);
    state1.cvar_M_HardwareMapDH_t := state0.cvar_M_HardwareMapDH_t + curDeltaSecs * derivcvar_M_HardwareMapDH_t(state0);
    state1.cvar_M_HardwareMapP_t := state0.cvar_M_HardwareMapP_t + curDeltaSecs * derivcvar_M_HardwareMapP_t(state0);
    state1.cvar_M_HardwareMapS_t := state0.cvar_M_HardwareMapS_t + curDeltaSecs * derivcvar_M_HardwareMapS_t(state0);
    state1.cvar_M_HardwareMapTB_t := state0.cvar_M_HardwareMapTB_t + curDeltaSecs * derivcvar_M_HardwareMapTB_t(state0);
    state1.cvar_M_STimer1_t := state0.cvar_M_STimer1_t + curDeltaSecs * derivcvar_M_STimer1_t(state0);
    state1.cvar_M_Timer1_t := state0.cvar_M_Timer1_t + curDeltaSecs * derivcvar_M_Timer1_t(state0);
    state1.cvar_M_TTimer1_t := state0.cvar_M_TTimer1_t + curDeltaSecs * derivcvar_M_TTimer1_t(state0);

    state0.curTime := curTime;
    state0.cvar_M_BTimer1_t := state1.cvar_M_BTimer1_t;
    state0.cvar_M_HardwareMapDH_t := state1.cvar_M_HardwareMapDH_t;
    state0.cvar_M_HardwareMapP_t := state1.cvar_M_HardwareMapP_t;
    state0.cvar_M_HardwareMapS_t := state1.cvar_M_HardwareMapS_t;
    state0.cvar_M_HardwareMapTB_t := state1.cvar_M_HardwareMapTB_t;
    state0.cvar_M_STimer1_t := state1.cvar_M_STimer1_t;
    state0.cvar_M_Timer1_t := state1.cvar_M_Timer1_t;
    state0.cvar_M_TTimer1_t := state1.cvar_M_TTimer1_t;
END_IF;

// Event loop.
WHILE TRUE DO
    progress := FALSE;

    // Event "A_airslide_c_off".
    IF NOT progress THEN
        b1 := (state0.dvar_M_sup_A_airslide) = (elit_On);
        b1 := b1 AND ((state0.dvar_M_sup_sup) = (elit_X));
        b1 := b1 AND ((state0.dvar_M_sup_S_elevator_down) = (elit_On));
        b1 := b1 AND ((state0.dvar_M_sup_S_Tinitialized) = (elit_On));
        IF b1 THEN
            progress := TRUE;
            state1 := state0;

            state1.dvar_M_sup_A_airslide := elit_Off;

            state0 := state1;
        END_IF;
    END_IF;

    // Event "A_airslide_c_on".
    IF NOT progress THEN
        b1 := (state0.dvar_M_sup_A_airslide) = (elit_Off);
        b1 := b1 AND ((state0.dvar_M_sup_sup) = (elit_X));
        b1 := b1 AND ((state0.dvar_M_sup_S_pusher) = (elit_On));
        b1 := b1 AND ((state0.dvar_M_sup_S_elevator_up) = (elit_On));
        b1 := b1 AND ((state0.dvar_M_sup_S_Tinitialized) = (elit_On));
        IF b1 THEN
            progress := TRUE;
            state1 := state0;

            state1.dvar_M_sup_A_airslide := elit_On;

            state0 := state1;
        END_IF;
    END_IF;

    // Event "A_bufferingready_c_off".
    IF NOT progress THEN
        b1 := (state0.dvar_M_sup_A_bufferingready) = (elit_On);
        b1 := b1 AND ((state0.dvar_M_sup_sup) = (elit_X));
        b1 := b1 AND ((state0.dvar_M_sup_S_Binitialized) = (elit_On));
        IF b1 THEN
            progress := TRUE;
            state1 := state0;

            state1.dvar_M_sup_A_bufferingready := elit_Off;

            state0 := state1;
        END_IF;
    END_IF;

    // Event "A_bufferingready_c_on".
    IF NOT progress THEN
        IF FALSE THEN
            progress := TRUE;
            state1 := state0;

            state1.dvar_M_sup_A_bufferingready := elit_On;

            state0 := state1;
        END_IF;
    END_IF;

    // Event "A_clamp_c_off".
    IF NOT progress THEN
        b1 := (state0.dvar_M_sup_A_clamp) = (elit_On);
        b1 := b1 AND ((state0.dvar_M_sup_ClampDrill) = (elit_eight));
        b1 := b1 AND ((state0.dvar_M_sup_sup) = (elit_X));
        b1 := b1 AND ((state0.dvar_M_sup_S_drill_up) = (elit_On));
        b1 := b1 AND ((state0.dvar_M_sup_S_Pinitialized) = (elit_On));
        IF b1 THEN
            progress := TRUE;
            state1 := state0;

            state1.dvar_M_sup_A_clamp := elit_Off;
            state1.dvar_M_sup_ClampDrill := elit_nine;

            state0 := state1;
        END_IF;
    END_IF;

    // Event "A_clamp_c_on".
    IF NOT progress THEN
        b1 := (state0.dvar_M_sup_A_clamp) = (elit_Off);
        b1 := b1 AND ((state0.dvar_M_sup_ClampDrill) = (elit_one2));
        b1 := b1 AND ((state0.dvar_M_sup_sup) = (elit_X));
        b1 := b1 AND ((state0.dvar_M_sup_A_turntable) = (elit_Off));
        b1 := b1 AND ((state0.dvar_M_sup_S_atdrill) = (elit_On));
        b1 := b1 AND ((state0.dvar_M_sup_S_Pinitialized) = (elit_On));
        b1 := b1 AND ((state0.dvar_M_sup_S_turntable) = (elit_On));
        b1 := b1 AND ((state0.dvar_M_sup_Timer) = (elit_Timeout));
        IF b1 THEN
            progress := TRUE;
            state1 := state0;

            state1.dvar_M_sup_A_clamp := elit_On;
            state1.dvar_M_sup_ClampDrill := elit_two2;

            state0 := state1;
        END_IF;
    END_IF;

    // Event "A_conveyer_c_off".
    IF NOT progress THEN
        b1 := (state0.dvar_M_sup_A_conveyer) = (elit_On);
        b1 := b1 AND ((state0.dvar_M_sup_sup) = (elit_X));
        b1 := b1 AND ((state0.dvar_M_sup_S_Sinitialized) = (elit_On));
        b1 := b1 AND ((state0.dvar_M_sup_S_slidefull) = (elit_On));
        IF b1 THEN
            progress := TRUE;
            state1 := state0;

            state1.dvar_M_sup_A_conveyer := elit_Off;

            state0 := state1;
        END_IF;
    END_IF;

    // Event "A_conveyer_c_on".
    IF NOT progress THEN
        b1 := (state0.dvar_M_sup_A_conveyer) = (elit_Off);
        b1 := b1 AND ((state0.dvar_M_sup_sup) = (elit_X));
        b1 := b1 AND ((state0.dvar_M_sup_S_product) = (elit_On));
        b1 := b1 AND ((state0.dvar_M_sup_S_Sinitialized) = (elit_On));
        IF b1 THEN
            progress := TRUE;
            state1 := state0;

            state1.dvar_M_sup_A_conveyer := elit_On;

            state0 := state1;
        END_IF;
    END_IF;

    // Event "A_conveyerB_c_off".
    IF NOT progress THEN
        b1 := (state0.dvar_M_sup_A_conveyerB) = (elit_On);
        b1 := b1 AND ((state0.dvar_M_sup_sup) = (elit_X));
        b1 := b1 AND ((state0.dvar_M_sup_BTimer) = (elit_Timeout));
        b1 := b1 AND ((state0.dvar_M_sup_S_Binitialized) = (elit_On));
        IF b1 THEN
            progress := TRUE;
            state1 := state0;

            state1.dvar_M_sup_A_conveyerB := elit_Off;

            state0 := state1;
        END_IF;
    END_IF;

    // Event "A_conveyerB_c_on".
    IF NOT progress THEN
        b1 := (state0.dvar_M_sup_A_conveyerB) = (elit_Off);
        b1 := b1 AND ((state0.dvar_M_sup_sup) = (elit_X));
        b1 := b1 AND ((state0.dvar_M_sup_S_atin) = (elit_On));
        b1 := b1 AND ((state0.dvar_M_sup_S_Binitialized) = (elit_On));
        IF b1 THEN
            progress := TRUE;
            state1 := state0;

            state1.dvar_M_sup_A_conveyerB := elit_On;

            state0 := state1;
        END_IF;
    END_IF;

    // Event "A_drill_c_off".
    IF NOT progress THEN
        b1 := (state0.dvar_M_sup_A_drill) = (elit_On);
        b1 := b1 AND ((state0.dvar_M_sup_ClampDrill) = (elit_seven));
        b1 := b1 AND ((state0.dvar_M_sup_sup) = (elit_X));
        b1 := b1 AND ((state0.dvar_M_sup_S_drill_down) = (elit_On));
        b1 := b1 AND ((state0.dvar_M_sup_S_Pinitialized) = (elit_On));
        IF b1 THEN
            progress := TRUE;
            state1 := state0;

            state1.dvar_M_sup_A_drill := elit_Off;
            state1.dvar_M_sup_ClampDrill := elit_eight;

            state0 := state1;
        END_IF;
    END_IF;

    // Event "A_drill_c_on".
    IF NOT progress THEN
        b1 := (state0.dvar_M_sup_A_drill) = (elit_Off);
        b1 := b1 AND ((state0.dvar_M_sup_ClampDrill) = (elit_two2));
        b1 := b1 AND ((state0.dvar_M_sup_sup) = (elit_X));
        b1 := b1 AND ((state0.dvar_M_sup_S_clamp) = (elit_On));
        b1 := b1 AND ((state0.dvar_M_sup_S_drill_up) = (elit_On));
        b1 := b1 AND ((state0.dvar_M_sup_S_Pinitialized) = (elit_On));
        IF b1 THEN
            progress := TRUE;
            state1 := state0;

            state1.dvar_M_sup_A_drill := elit_On;
            state1.dvar_M_sup_ClampDrill := elit_three2;

            state0 := state1;
        END_IF;
    END_IF;

    // Event "A_drilldown_c_off".
    IF NOT progress THEN
        b1 := (state0.dvar_M_sup_A_drilldown) = (elit_On);
        b1 := b1 AND ((state0.dvar_M_sup_ClampDrill) = (elit_five));
        b1 := b1 AND ((state0.dvar_M_sup_sup) = (elit_X));
        b1 := b1 AND ((state0.dvar_M_sup_S_drill_down) = (elit_On));
        IF b1 THEN
            progress := TRUE;
            state1 := state0;

            state1.dvar_M_sup_A_drilldown := elit_Off;
            state1.dvar_M_sup_ClampDrill := elit_six;

            state0 := state1;
        END_IF;
    END_IF;

    // Event "A_drilldown_c_on".
    IF NOT progress THEN
        b1 := (state0.dvar_M_sup_A_drilldown) = (elit_Off);
        b1 := b1 AND ((state0.dvar_M_sup_ClampDrill) = (elit_four2));
        b1 := b1 AND ((state0.dvar_M_sup_sup) = (elit_X));
        b1 := b1 AND ((state0.dvar_M_sup_S_drill_up) = (elit_On));
        b1 := b1 AND ((state0.dvar_M_sup_S_Pinitialized) = (elit_On));
        IF b1 THEN
            progress := TRUE;
            state1 := state0;

            state1.dvar_M_sup_A_drilldown := elit_On;
            state1.dvar_M_sup_ClampDrill := elit_five;

            state0 := state1;
        END_IF;
    END_IF;

    // Event "A_drillup_c_off".
    IF NOT progress THEN
        b1 := (state0.dvar_M_sup_A_drillup) = (elit_On);
        b1 := b1 AND ((state0.dvar_M_sup_ClampDrill) = (elit_three2));
        b1 := b1 AND ((state0.dvar_M_sup_sup) = (elit_X));
        b1 := b1 AND ((state0.dvar_M_sup_S_drill_up) = (elit_On));
        b1 := b1 AND ((state0.dvar_M_sup_S_Pinitialized) = (elit_On));
        IF b1 THEN
            progress := TRUE;
            state1 := state0;

            state1.dvar_M_sup_A_drillup := elit_Off;
            state1.dvar_M_sup_ClampDrill := elit_four2;

            state0 := state1;
        END_IF;
    END_IF;

    // Event "A_drillup_c_on".
    IF NOT progress THEN
        b1 := (state0.dvar_M_sup_A_drillup) = (elit_Off);
        b1 := b1 AND ((state0.dvar_M_sup_ClampDrill) = (elit_six));
        b1 := b1 AND ((state0.dvar_M_sup_sup) = (elit_X));
        b1 := b1 AND ((state0.dvar_M_sup_S_drill_down) = (elit_On));
        IF b1 THEN
            progress := TRUE;
            state1 := state0;

            state1.dvar_M_sup_A_drillup := elit_On;
            state1.dvar_M_sup_ClampDrill := elit_seven;

            state0 := state1;
        END_IF;
    END_IF;

    // Event "A_eject_c_off".
    IF NOT progress THEN
        b1 := (state0.dvar_M_sup_A_eject) = (elit_On);
        b1 := b1 AND ((state0.dvar_M_sup_sup) = (elit_X));
        b1 := b1 AND ((state0.dvar_M_sup_A_conveyer) = (elit_Off));
        b1 := b1 AND ((state0.dvar_M_sup_S_atexit) = (elit_Off));
        b1 := b1 AND ((state0.dvar_M_sup_S_Pinitialized) = (elit_On));
        IF b1 THEN
            progress := TRUE;
            state1 := state0;

            state1.dvar_M_sup_A_eject := elit_Off;

            state0 := state1;
        END_IF;
    END_IF;

    // Event "A_eject_c_on".
    IF NOT progress THEN
        b1 := (state0.dvar_M_sup_A_eject) = (elit_Off);
        b1 := b1 AND ((state0.dvar_M_sup_sup) = (elit_X));
        b1 := b1 AND ((state0.dvar_M_sup_A_turntable) = (elit_Off));
        b1 := b1 AND ((state0.dvar_M_sup_S_atexit) = (elit_On));
        b1 := b1 AND ((state0.dvar_M_sup_S_Pinitialized) = (elit_On));
        b1 := b1 AND ((state0.dvar_M_sup_S_turntable) = (elit_On));
        b1 := b1 AND ((state0.dvar_M_sup_Timer) = (elit_Timeout));
        IF b1 THEN
            progress := TRUE;
            state1 := state0;

            state1.dvar_M_sup_A_eject := elit_On;

            state0 := state1;
        END_IF;
    END_IF;

    // Event "A_ejectpulse_c_off".
    IF NOT progress THEN
        b1 := (state0.dvar_M_sup_A_ejectpulse) = (elit_On);
        b1 := b1 AND ((state0.dvar_M_sup_sup) = (elit_X));
        b1 := b1 AND ((state0.dvar_M_sup_S_Hinitialized) = (elit_On));
        b1 := b1 AND ((state0.dvar_M_sup_S_vacuum) = (elit_Off));
        IF b1 THEN
            progress := TRUE;
            state1 := state0;

            state1.dvar_M_sup_A_ejectpulse := elit_Off;

            state0 := state1;
        END_IF;
    END_IF;

    // Event "A_ejectpulse_c_on".
    IF NOT progress THEN
        b1 := (state0.dvar_M_sup_A_ejectpulse) = (elit_Off);
        b1 := b1 AND ((state0.dvar_M_sup_sup) = (elit_X));
        b1 := b1 AND ((state0.dvar_M_sup_S_Hinitialized) = (elit_On));
        b1 := b1 AND ((state0.dvar_M_sup_S_transfer_atdrop) = (elit_On));
        b1 := b1 AND ((state0.dvar_M_sup_S_vacuum) = (elit_On));
        IF b1 THEN
            progress := TRUE;
            state1 := state0;

            state1.dvar_M_sup_A_ejectpulse := elit_On;

            state0 := state1;
        END_IF;
    END_IF;

    // Event "A_elevator_down_c_off".
    IF NOT progress THEN
        b1 := (state0.dvar_M_sup_A_elevator_down) = (elit_On);
        b1 := b1 AND ((state0.dvar_M_sup_PusherLift) = (elit_One));
        b1 := b1 AND ((state0.dvar_M_sup_sup) = (elit_X));
        b1 := b1 AND ((state0.dvar_M_sup_S_pusher) = (elit_Off));
        b1 := b1 AND ((state0.dvar_M_sup_S_elevator_down) = (elit_On));
        b1 := b1 AND ((state0.dvar_M_sup_S_reflective) = (elit_Off));
        b1 := b1 AND ((state0.dvar_M_sup_S_capacitive) = (elit_On));
        b1 := b1 AND ((state0.dvar_M_sup_S_transfer_athalfway) = (elit_On));
        b1 := b1 AND ((state0.dvar_M_sup_S_Tinitialized) = (elit_On));
        b1 := b1 AND ((state0.dvar_M_sup_TTimer) = (elit_Timeout));
        IF b1 THEN
            progress := TRUE;
            state1 := state0;

            state1.dvar_M_sup_A_elevator_down := elit_Off;
            state1.dvar_M_sup_PusherLift := elit_Two;

            state0 := state1;
        END_IF;
    END_IF;

    // Event "A_elevator_down_c_on".
    IF NOT progress THEN
        b1 := (state0.dvar_M_sup_A_elevator_down) = (elit_Off);
        b1 := b1 AND ((state0.dvar_M_sup_PusherLift) = (elit_Four));
        b1 := b1 AND ((state0.dvar_M_sup_sup) = (elit_X));
        b1 := b1 AND ((state0.dvar_M_sup_A_elevator_up) = (elit_Off));
        b1 := b1 AND ((state0.dvar_M_sup_S_opticalT) = (elit_Off));
        b1 := b1 AND ((state0.dvar_M_sup_S_pusher) = (elit_Off));
        b1 := b1 AND ((state0.dvar_M_sup_S_elevator_up) = (elit_On));
        b1 := b1 AND ((state0.dvar_M_sup_S_Tinitialized) = (elit_On));
        b1 := b1 AND ((state0.dvar_M_sup_TTimer) = (elit_Timeout));
        IF b1 THEN
            progress := TRUE;
            state1 := state0;

            state1.dvar_M_sup_A_elevator_down := elit_On;
            state1.dvar_M_sup_PusherLift := elit_One;

            state0 := state1;
        END_IF;
    END_IF;

    // Event "A_elevator_up_c_off".
    IF NOT progress THEN
        b1 := (state0.dvar_M_sup_A_elevator_up) = (elit_On);
        b1 := b1 AND ((state0.dvar_M_sup_sup) = (elit_X));
        b1 := b1 AND ((state0.dvar_M_sup_S_opticalT) = (elit_Off));
        b1 := b1 AND ((state0.dvar_M_sup_S_pusher) = (elit_Off));
        b1 := b1 AND ((state0.dvar_M_sup_S_elevator_up) = (elit_On));
        b1 := b1 AND ((state0.dvar_M_sup_S_Tinitialized) = (elit_On));
        b1 := b1 AND ((state0.dvar_M_sup_TTimer) = (elit_Timeout));
        IF b1 THEN
            progress := TRUE;
            state1 := state0;

            state1.dvar_M_sup_A_elevator_up := elit_Off;

            state0 := state1;
        END_IF;
    END_IF;

    // Event "A_elevator_up_c_on".
    IF NOT progress THEN
        b1 := (state0.dvar_M_sup_A_elevator_up) = (elit_Off);
        b1 := b1 AND ((state0.dvar_M_sup_sup) = (elit_X));
        b1 := b1 AND ((state0.dvar_M_sup_A_elevator_down) = (elit_Off));
        b1 := b1 AND ((state0.dvar_M_sup_S_pusher) = (elit_Off));
        b1 := b1 AND ((state0.dvar_M_sup_S_elevator_down) = (elit_On));
        b1 := b1 AND ((state0.dvar_M_sup_S_reflective) = (elit_Off));
        b1 := b1 AND ((state0.dvar_M_sup_S_capacitive) = (elit_On));
        b1 := b1 AND ((state0.dvar_M_sup_S_transfer_athalfway) = (elit_On));
        b1 := b1 AND ((state0.dvar_M_sup_S_Tinitialized) = (elit_On));
        b1 := b1 AND ((state0.dvar_M_sup_TTimer) = (elit_Timeout));
        IF b1 THEN
            progress := TRUE;
            state1 := state0;

            state1.dvar_M_sup_A_elevator_up := elit_On;

            state0 := state1;
        END_IF;
    END_IF;

    // Event "A_gate1_c_off".
    IF NOT progress THEN
        b1 := (state0.dvar_M_sup_A_gate1) = (elit_On);
        b1 := b1 AND ((state0.dvar_M_sup_sup) = (elit_X));
        b1 := b1 AND ((state0.dvar_M_sup_A_stopperretract) = (elit_Off));
        b1 := b1 AND ((state0.dvar_M_sup_S_Sinitialized) = (elit_On));
        b1 := b1 AND ((state0.dvar_M_sup_S_slidefull) = (elit_On));
        IF b1 THEN
            progress := TRUE;
            state1 := state0;

            state1.dvar_M_sup_A_gate1 := elit_Off;

            state0 := state1;
        END_IF;
    END_IF;

    // Event "A_gate1_c_on".
    IF NOT progress THEN
        b1 := (state0.dvar_M_sup_A_gate1) = (elit_Off);
        b1 := b1 AND ((state0.dvar_M_sup_sup) = (elit_X));
        b1 := b1 AND ((state0.dvar_M_sup_A_stopperretract) = (elit_Off));
        b1 := b1 AND ((state0.dvar_M_sup_S_inductive) = (elit_Off));
        b1 := b1 AND ((state0.dvar_M_sup_S_optical) = (elit_On));
        b1 := b1 AND ((state0.dvar_M_sup_S_Sinitialized) = (elit_On));
        b1 := b1 AND ((state0.dvar_M_sup_STimer) = (elit_Timeout));
        IF b1 THEN
            progress := TRUE;
            state1 := state0;

            state1.dvar_M_sup_A_gate1 := elit_On;

            state0 := state1;
        END_IF;
    END_IF;

    // Event "A_gate2_c_off".
    IF NOT progress THEN
        b1 := (state0.dvar_M_sup_A_gate2) = (elit_On);
        b1 := b1 AND ((state0.dvar_M_sup_sup) = (elit_X));
        b1 := b1 AND ((state0.dvar_M_sup_A_stopperretract) = (elit_Off));
        b1 := b1 AND ((state0.dvar_M_sup_S_Sinitialized) = (elit_On));
        b1 := b1 AND ((state0.dvar_M_sup_S_slidefull) = (elit_On));
        IF b1 THEN
            progress := TRUE;
            state1 := state0;

            state1.dvar_M_sup_A_gate2 := elit_Off;

            state0 := state1;
        END_IF;
    END_IF;

    // Event "A_gate2_c_on".
    IF NOT progress THEN
        b1 := (state0.dvar_M_sup_A_gate2) = (elit_Off);
        b1 := b1 AND ((state0.dvar_M_sup_sup) = (elit_X));
        b1 := b1 AND ((state0.dvar_M_sup_A_stopperretract) = (elit_Off));
        b1 := b1 AND ((state0.dvar_M_sup_S_inductive) = (elit_On));
        b1 := b1 AND ((state0.dvar_M_sup_S_optical) = (elit_On));
        b1 := b1 AND ((state0.dvar_M_sup_S_Sinitialized) = (elit_On));
        b1 := b1 AND ((state0.dvar_M_sup_STimer) = (elit_Timeout));
        IF b1 THEN
            progress := TRUE;
            state1 := state0;

            state1.dvar_M_sup_A_gate2 := elit_On;

            state0 := state1;
        END_IF;
    END_IF;

    // Event "A_gripperclose_c_off".
    IF NOT progress THEN
        b1 := (state0.dvar_M_sup_A_gripperclose) = (elit_On);
        b1 := b1 AND ((state0.dvar_M_sup_sup) = (elit_X));
        b1 := b1 AND ((state0.dvar_M_sup_S_Hinitialized) = (elit_On));
        b1 := b1 AND ((state0.dvar_M_sup_S_xpos_atdrop) = (elit_On));
        b1 := b1 AND ((state0.dvar_M_sup_S_zpos_atdown) = (elit_On));
        IF b1 THEN
            progress := TRUE;
            state1 := state0;

            state1.dvar_M_sup_A_gripperclose := elit_Off;

            state0 := state1;
        END_IF;
    END_IF;

    // Event "A_gripperclose_c_on".
    IF NOT progress THEN
        b1 := (state0.dvar_M_sup_A_gripperclose) = (elit_Off);
        b1 := b1 AND ((state0.dvar_M_sup_sup) = (elit_X));
        IF b1 THEN
            b3 := (state0.dvar_M_sup_S_Hinitialized) = (elit_On);
            b3 := b3 AND ((state0.dvar_M_sup_S_xpos_at3) = (elit_On));
            b3 := b3 AND ((state0.dvar_M_sup_S_zpos_atdown) = (elit_On));
            b2 := b3;
            IF NOT(b2) THEN
                b3 := (state0.dvar_M_sup_S_Hinitialized) = (elit_On);
                b3 := b3 AND ((state0.dvar_M_sup_S_xpos_at3) = (elit_Off));
                b3 := b3 AND ((state0.dvar_M_sup_S_xpos_at2) = (elit_On));
                b3 := b3 AND ((state0.dvar_M_sup_S_zpos_atdown) = (elit_On));
                b2 := b2 OR (b3);
            END_IF;
            IF NOT(b2) THEN
                b3 := (state0.dvar_M_sup_S_Hinitialized) = (elit_On);
                b3 := b3 AND ((state0.dvar_M_sup_S_xpos_at3) = (elit_Off));
                b3 := b3 AND ((state0.dvar_M_sup_S_xpos_at2) = (elit_Off));
                b3 := b3 AND ((state0.dvar_M_sup_S_xpos_at1) = (elit_On));
                b3 := b3 AND ((state0.dvar_M_sup_S_zpos_atdown) = (elit_On));
                b2 := b2 OR (b3);
            END_IF;
            b1 := b1 AND (b2);
        END_IF;
        IF b1 THEN
            progress := TRUE;
            state1 := state0;

            state1.dvar_M_sup_A_gripperclose := elit_On;

            state0 := state1;
        END_IF;
    END_IF;

    // Event "A_handlingready_c_off".
    IF NOT progress THEN
        b1 := (state0.dvar_M_sup_A_handlingready) = (elit_On);
        b1 := b1 AND ((state0.dvar_M_sup_sup) = (elit_X));
        b1 := b1 AND ((state0.dvar_M_sup_S_Hinitialized) = (elit_On));
        IF b1 THEN
            progress := TRUE;
            state1 := state0;

            state1.dvar_M_sup_A_handlingready := elit_Off;

            state0 := state1;
        END_IF;
    END_IF;

    // Event "A_handlingready_c_on".
    IF NOT progress THEN
        IF FALSE THEN
            progress := TRUE;
            state1 := state0;

            state1.dvar_M_sup_A_handlingready := elit_On;

            state0 := state1;
        END_IF;
    END_IF;

    // Event "A_processingready_c_off".
    IF NOT progress THEN
        b1 := (state0.dvar_M_sup_A_processingready) = (elit_On);
        b1 := b1 AND ((state0.dvar_M_sup_sup) = (elit_X));
        b1 := b1 AND ((state0.dvar_M_sup_S_Pinitialized) = (elit_On));
        IF b1 THEN
            progress := TRUE;
            state1 := state0;

            state1.dvar_M_sup_A_processingready := elit_Off;

            state0 := state1;
        END_IF;
    END_IF;

    // Event "A_processingready_c_on".
    IF NOT progress THEN
        IF FALSE THEN
            progress := TRUE;
            state1 := state0;

            state1.dvar_M_sup_A_processingready := elit_On;

            state0 := state1;
        END_IF;
    END_IF;

    // Event "A_pusher_c_off".
    IF NOT progress THEN
        b1 := (state0.dvar_M_sup_A_pusher) = (elit_On);
        b1 := b1 AND ((state0.dvar_M_sup_PusherLift) = (elit_Three));
        b1 := b1 AND ((state0.dvar_M_sup_sup) = (elit_X));
        b1 := b1 AND ((state0.dvar_M_sup_S_pusher) = (elit_On));
        b1 := b1 AND ((state0.dvar_M_sup_S_Tinitialized) = (elit_On));
        IF b1 THEN
            progress := TRUE;
            state1 := state0;

            state1.dvar_M_sup_A_pusher := elit_Off;
            state1.dvar_M_sup_PusherLift := elit_Four;

            state0 := state1;
        END_IF;
    END_IF;

    // Event "A_pusher_c_on".
    IF NOT progress THEN
        b1 := (state0.dvar_M_sup_A_pusher) = (elit_Off);
        b1 := b1 AND ((state0.dvar_M_sup_PusherLift) = (elit_Two));
        b1 := b1 AND ((state0.dvar_M_sup_sup) = (elit_X));
        b1 := b1 AND ((state0.dvar_M_sup_S_elevator_up) = (elit_On));
        b1 := b1 AND ((state0.dvar_M_sup_S_Tinitialized) = (elit_On));
        IF b1 THEN
            progress := TRUE;
            state1 := state0;

            state1.dvar_M_sup_A_pusher := elit_On;
            state1.dvar_M_sup_PusherLift := elit_Three;

            state0 := state1;
        END_IF;
    END_IF;

    // Event "A_pusher1_c_off".
    IF NOT progress THEN
        b1 := (state0.dvar_M_sup_A_pusher1) = (elit_On);
        b1 := b1 AND ((state0.dvar_M_sup_sup) = (elit_X));
        b1 := b1 AND ((state0.dvar_M_sup_S_Dinitialized) = (elit_On));
        b1 := b1 AND ((state0.dvar_M_sup_S_pusher1_out) = (elit_On));
        b1 := b1 AND ((state0.dvar_M_sup_S_stack1_filled) = (elit_On));
        b1 := b1 AND ((state0.dvar_M_sup_S_product1) = (elit_Off));
        IF b1 THEN
            progress := TRUE;
            state1 := state0;

            state1.dvar_M_sup_A_pusher1 := elit_Off;

            state0 := state1;
        END_IF;
    END_IF;

    // Event "A_pusher1_c_on".
    IF NOT progress THEN
        b1 := (state0.dvar_M_sup_A_pusher1) = (elit_Off);
        b1 := b1 AND ((state0.dvar_M_sup_sup) = (elit_X));
        b1 := b1 AND ((state0.dvar_M_sup_S_Dinitialized) = (elit_On));
        b1 := b1 AND ((state0.dvar_M_sup_S_pusher1_in) = (elit_On));
        b1 := b1 AND ((state0.dvar_M_sup_S_product1) = (elit_Off));
        IF b1 THEN
            progress := TRUE;
            state1 := state0;

            state1.dvar_M_sup_A_pusher1 := elit_On;

            state0 := state1;
        END_IF;
    END_IF;

    // Event "A_pusher2_c_off".
    IF NOT progress THEN
        b1 := (state0.dvar_M_sup_A_pusher2) = (elit_On);
        b1 := b1 AND ((state0.dvar_M_sup_sup) = (elit_X));
        b1 := b1 AND ((state0.dvar_M_sup_S_Dinitialized) = (elit_On));
        b1 := b1 AND ((state0.dvar_M_sup_S_pusher2_out) = (elit_On));
        b1 := b1 AND ((state0.dvar_M_sup_S_product2) = (elit_Off));
        b1 := b1 AND ((state0.dvar_M_sup_S_stack2_filled) = (elit_On));
        IF b1 THEN
            progress := TRUE;
            state1 := state0;

            state1.dvar_M_sup_A_pusher2 := elit_Off;

            state0 := state1;
        END_IF;
    END_IF;

    // Event "A_pusher2_c_on".
    IF NOT progress THEN
        b1 := (state0.dvar_M_sup_A_pusher2) = (elit_Off);
        b1 := b1 AND ((state0.dvar_M_sup_sup) = (elit_X));
        b1 := b1 AND ((state0.dvar_M_sup_S_Dinitialized) = (elit_On));
        b1 := b1 AND ((state0.dvar_M_sup_S_pusher2_in) = (elit_On));
        b1 := b1 AND ((state0.dvar_M_sup_S_product2) = (elit_Off));
        IF b1 THEN
            progress := TRUE;
            state1 := state0;

            state1.dvar_M_sup_A_pusher2 := elit_On;

            state0 := state1;
        END_IF;
    END_IF;

    // Event "A_pusher3_c_off".
    IF NOT progress THEN
        b1 := (state0.dvar_M_sup_A_pusher3) = (elit_On);
        b1 := b1 AND ((state0.dvar_M_sup_sup) = (elit_X));
        b1 := b1 AND ((state0.dvar_M_sup_S_Dinitialized) = (elit_On));
        b1 := b1 AND ((state0.dvar_M_sup_S_pusher3_out) = (elit_On));
        b1 := b1 AND ((state0.dvar_M_sup_S_product3) = (elit_Off));
        b1 := b1 AND ((state0.dvar_M_sup_S_stack3_filled) = (elit_On));
        IF b1 THEN
            progress := TRUE;
            state1 := state0;

            state1.dvar_M_sup_A_pusher3 := elit_Off;

            state0 := state1;
        END_IF;
    END_IF;

    // Event "A_pusher3_c_on".
    IF NOT progress THEN
        b1 := (state0.dvar_M_sup_A_pusher3) = (elit_Off);
        b1 := b1 AND ((state0.dvar_M_sup_sup) = (elit_X));
        b1 := b1 AND ((state0.dvar_M_sup_S_Dinitialized) = (elit_On));
        b1 := b1 AND ((state0.dvar_M_sup_S_pusher3_in) = (elit_On));
        b1 := b1 AND ((state0.dvar_M_sup_S_product3) = (elit_Off));
        IF b1 THEN
            progress := TRUE;
            state1 := state0;

            state1.dvar_M_sup_A_pusher3 := elit_On;

            state0 := state1;
        END_IF;
    END_IF;

    // Event "A_separator_c_off".
    IF NOT progress THEN
        b1 := (state0.dvar_M_sup_A_separator) = (elit_On);
        b1 := b1 AND ((state0.dvar_M_sup_sup) = (elit_X));
        b1 := b1 AND ((state0.dvar_M_sup_S_atinput) = (elit_Off));
        b1 := b1 AND ((state0.dvar_M_sup_S_atseparator) = (elit_Off));
        b1 := b1 AND ((state0.dvar_M_sup_S_Binitialized) = (elit_On));
        b1 := b1 AND ((state0.dvar_M_sup_S_separator_opened) = (elit_On));
        b1 := b1 AND ((state0.dvar_M_sup_S_turntable) = (elit_On));
        IF b1 THEN
            progress := TRUE;
            state1 := state0;

            state1.dvar_M_sup_A_separator := elit_Off;

            state0 := state1;
        END_IF;
    END_IF;

    // Event "A_separator_c_on".
    IF NOT progress THEN
        b1 := (state0.dvar_M_sup_A_separator) = (elit_Off);
        b1 := b1 AND ((state0.dvar_M_sup_sup) = (elit_X));
        b1 := b1 AND ((state0.dvar_M_sup_S_atseparator) = (elit_On));
        b1 := b1 AND ((state0.dvar_M_sup_S_Binitialized) = (elit_On));
        b1 := b1 AND ((state0.dvar_M_sup_S_separator_closed) = (elit_On));
        IF b1 THEN
            progress := TRUE;
            state1 := state0;

            state1.dvar_M_sup_A_separator := elit_On;

            state0 := state1;
        END_IF;
    END_IF;

    // Event "A_sortingready_c_off".
    IF NOT progress THEN
        b1 := (state0.dvar_M_sup_A_sortingready) = (elit_On);
        b1 := b1 AND ((state0.dvar_M_sup_sup) = (elit_X));
        b1 := b1 AND ((state0.dvar_M_sup_S_Sinitialized) = (elit_On));
        IF b1 THEN
            progress := TRUE;
            state1 := state0;

            state1.dvar_M_sup_A_sortingready := elit_Off;

            state0 := state1;
        END_IF;
    END_IF;

    // Event "A_sortingready_c_on".
    IF NOT progress THEN
        IF FALSE THEN
            progress := TRUE;
            state1 := state0;

            state1.dvar_M_sup_A_sortingready := elit_On;

            state0 := state1;
        END_IF;
    END_IF;

    // Event "A_stopperretract_c_off".
    IF NOT progress THEN
        b1 := (state0.dvar_M_sup_A_stopperretract) = (elit_On);
        b1 := b1 AND ((state0.dvar_M_sup_sup) = (elit_X));
        b1 := b1 AND ((state0.dvar_M_sup_S_Sinitialized) = (elit_On));
        b1 := b1 AND ((state0.dvar_M_sup_S_slidefull) = (elit_On));
        IF b1 THEN
            progress := TRUE;
            state1 := state0;

            state1.dvar_M_sup_A_stopperretract := elit_Off;

            state0 := state1;
        END_IF;
    END_IF;

    // Event "A_stopperretract_c_on".
    IF NOT progress THEN
        b1 := (state0.dvar_M_sup_A_stopperretract) = (elit_Off);
        b1 := b1 AND ((state0.dvar_M_sup_sup) = (elit_X));
        b1 := b1 AND ((state0.dvar_M_sup_S_Sinitialized) = (elit_On));
        b1 := b1 AND ((state0.dvar_M_sup_S_slidefull) = (elit_Off));
        b1 := b1 AND ((state0.dvar_M_sup_STimer) = (elit_Timeout));
        IF b1 THEN
            progress := TRUE;
            state1 := state0;

            state1.dvar_M_sup_A_stopperretract := elit_On;

            state0 := state1;
        END_IF;
    END_IF;

    // Event "A_tester_c_off".
    IF NOT progress THEN
        b1 := (state0.dvar_M_sup_A_tester) = (elit_On);
        b1 := b1 AND ((state0.dvar_M_sup_sup) = (elit_X));
        b1 := b1 AND ((state0.dvar_M_sup_S_Pinitialized) = (elit_On));
        b1 := b1 AND ((state0.dvar_M_sup_S_test_ok) = (elit_On));
        b1 := b1 AND ((state0.dvar_M_sup_Tester) = (elit_Two));
        IF b1 THEN
            progress := TRUE;
            state1 := state0;

            state1.dvar_M_sup_A_tester := elit_Off;
            state1.dvar_M_sup_Tester := elit_Three;

            state0 := state1;
        END_IF;
    END_IF;

    // Event "A_tester_c_on".
    IF NOT progress THEN
        b1 := (state0.dvar_M_sup_A_tester) = (elit_Off);
        b1 := b1 AND ((state0.dvar_M_sup_sup) = (elit_X));
        b1 := b1 AND ((state0.dvar_M_sup_A_turntable) = (elit_Off));
        b1 := b1 AND ((state0.dvar_M_sup_S_attest) = (elit_On));
        b1 := b1 AND ((state0.dvar_M_sup_S_Pinitialized) = (elit_On));
        b1 := b1 AND ((state0.dvar_M_sup_S_turntable) = (elit_On));
        b1 := b1 AND ((state0.dvar_M_sup_Timer) = (elit_Timeout));
        b1 := b1 AND ((state0.dvar_M_sup_Tester) = (elit_One));
        IF b1 THEN
            progress := TRUE;
            state1 := state0;

            state1.dvar_M_sup_A_tester := elit_On;
            state1.dvar_M_sup_Tester := elit_Two;

            state0 := state1;
        END_IF;
    END_IF;

    // Event "A_testingready_c_off".
    IF NOT progress THEN
        IF FALSE THEN
            progress := TRUE;
            state1 := state0;

            state1.dvar_M_sup_A_testingready := elit_Off;

            state0 := state1;
        END_IF;
    END_IF;

    // Event "A_testingready_c_on".
    IF NOT progress THEN
        IF FALSE THEN
            progress := TRUE;
            state1 := state0;

            state1.dvar_M_sup_A_testingready := elit_On;

            state0 := state1;
        END_IF;
    END_IF;

    // Event "A_transfer2droppos_c_off".
    IF NOT progress THEN
        b1 := (state0.dvar_M_sup_A_transfer2droppos) = (elit_On);
        b1 := b1 AND ((state0.dvar_M_sup_sup) = (elit_X));
        IF b1 THEN
            b2 := (state0.dvar_M_sup_S_Hinitialized) = (elit_Off);
            b2 := b2 OR ((state0.dvar_M_sup_S_elevator_down) = (elit_Off));
            b2 := b2 OR ((state0.dvar_M_sup_S_capacitive) = (elit_Off));
            b2 := b2 OR ((state0.dvar_M_sup_S_transfer_athalfway) = (elit_On));
            b2 := b2 OR ((state0.dvar_M_sup_S_transfer_atdrop) = (elit_On));
            b1 := b1 AND (b2);
        END_IF;
        IF b1 THEN
            b2 := (state0.dvar_M_sup_S_Hinitialized) = (elit_Off);
            b2 := b2 OR ((state0.dvar_M_sup_S_elevator_down) = (elit_Off));
            b2 := b2 OR ((state0.dvar_M_sup_S_capacitive) = (elit_On));
            b2 := b2 OR ((state0.dvar_M_sup_S_transfer_atdrop) = (elit_On));
            b1 := b1 AND (b2);
        END_IF;
        IF b1 THEN
            b2 := (state0.dvar_M_sup_S_Hinitialized) = (elit_Off);
            b2 := b2 OR ((state0.dvar_M_sup_S_elevator_down) = (elit_On));
            b2 := b2 OR ((state0.dvar_M_sup_S_transfer_athalfway) = (elit_On));
            b2 := b2 OR ((state0.dvar_M_sup_S_transfer_atdrop) = (elit_On));
            b1 := b1 AND (b2);
        END_IF;
        b1 := b1 AND ((state0.dvar_M_sup_S_Hinitialized) = (elit_On));
        IF b1 THEN
            progress := TRUE;
            state1 := state0;

            state1.dvar_M_sup_A_transfer2droppos := elit_Off;

            state0 := state1;
        END_IF;
    END_IF;

    // Event "A_transfer2droppos_c_on".
    IF NOT progress THEN
        b1 := (state0.dvar_M_sup_A_transfer2droppos) = (elit_Off);
        b1 := b1 AND ((state0.dvar_M_sup_sup) = (elit_X));
        IF b1 THEN
            b3 := (state0.dvar_M_sup_A_transfer2pickpos) = (elit_Off);
            b3 := b3 AND ((state0.dvar_M_sup_S_Hinitialized) = (elit_On));
            b3 := b3 AND ((state0.dvar_M_sup_S_elevator_down) = (elit_On));
            b3 := b3 AND ((state0.dvar_M_sup_S_capacitive) = (elit_On));
            b3 := b3 AND ((state0.dvar_M_sup_S_transfer_atpickup) = (elit_On));
            b3 := b3 AND ((state0.dvar_M_sup_S_vacuum) = (elit_On));
            b2 := b3;
            IF NOT(b2) THEN
                b3 := (state0.dvar_M_sup_A_transfer2pickpos) = (elit_Off);
                b3 := b3 AND ((state0.dvar_M_sup_S_Hinitialized) = (elit_On));
                b3 := b3 AND ((state0.dvar_M_sup_S_elevator_down) = (elit_On));
                b3 := b3 AND ((state0.dvar_M_sup_S_capacitive) = (elit_Off));
                b3 := b3 AND ((state0.dvar_M_sup_S_transfer_atpickup) = (elit_On));
                b3 := b3 AND ((state0.dvar_M_sup_S_vacuum) = (elit_On));
                b2 := b2 OR (b3);
            END_IF;
            IF NOT(b2) THEN
                b3 := (state0.dvar_M_sup_A_transfer2pickpos) = (elit_Off);
                b3 := b3 AND ((state0.dvar_M_sup_S_Hinitialized) = (elit_On));
                b3 := b3 AND ((state0.dvar_M_sup_S_elevator_down) = (elit_On));
                b3 := b3 AND ((state0.dvar_M_sup_S_capacitive) = (elit_Off));
                b3 := b3 AND ((state0.dvar_M_sup_S_transfer_atpickup) = (elit_Off));
                b3 := b3 AND ((state0.dvar_M_sup_S_transfer_athalfway) = (elit_On));
                b3 := b3 AND ((state0.dvar_M_sup_S_vacuum) = (elit_On));
                b2 := b2 OR (b3);
            END_IF;
            IF NOT(b2) THEN
                b3 := (state0.dvar_M_sup_A_transfer2pickpos) = (elit_Off);
                b3 := b3 AND ((state0.dvar_M_sup_S_Hinitialized) = (elit_On));
                b3 := b3 AND ((state0.dvar_M_sup_S_elevator_down) = (elit_Off));
                b3 := b3 AND ((state0.dvar_M_sup_S_transfer_atpickup) = (elit_On));
                b3 := b3 AND ((state0.dvar_M_sup_S_vacuum) = (elit_On));
                b2 := b2 OR (b3);
            END_IF;
            b1 := b1 AND (b2);
        END_IF;
        IF b1 THEN
            progress := TRUE;
            state1 := state0;

            state1.dvar_M_sup_A_transfer2droppos := elit_On;

            state0 := state1;
        END_IF;
    END_IF;

    // Event "A_transfer2pickpos_c_off".
    IF NOT progress THEN
        b1 := (state0.dvar_M_sup_A_transfer2pickpos) = (elit_On);
        b1 := b1 AND ((state0.dvar_M_sup_sup) = (elit_X));
        IF b1 THEN
            b3 := (state0.dvar_M_sup_S_Hinitialized) = (elit_On);
            b3 := b3 AND ((state0.dvar_M_sup_S_transfer_atpickup) = (elit_On));
            b2 := b3;
            IF NOT(b2) THEN
                b3 := (state0.dvar_M_sup_S_Hinitialized) = (elit_On);
                b3 := b3 AND ((state0.dvar_M_sup_S_transfer_atpickup) = (elit_Off));
                b3 := b3 AND ((state0.dvar_M_sup_S_transfer_athalfway) = (elit_On));
                b3 := b3 AND ((state0.dvar_M_sup_S_product4) = (elit_Off));
                b2 := b2 OR (b3);
            END_IF;
            b1 := b1 AND (b2);
        END_IF;
        IF b1 THEN
            progress := TRUE;
            state1 := state0;

            state1.dvar_M_sup_A_transfer2pickpos := elit_Off;

            state0 := state1;
        END_IF;
    END_IF;

    // Event "A_transfer2pickpos_c_on".
    IF NOT progress THEN
        b1 := (state0.dvar_M_sup_A_transfer2pickpos) = (elit_Off);
        b1 := b1 AND ((state0.dvar_M_sup_sup) = (elit_X));
        IF b1 THEN
            b3 := (state0.dvar_M_sup_A_transfer2droppos) = (elit_Off);
            b3 := b3 AND ((state0.dvar_M_sup_S_Hinitialized) = (elit_On));
            b3 := b3 AND ((state0.dvar_M_sup_S_transfer_athalfway) = (elit_On));
            b3 := b3 AND ((state0.dvar_M_sup_S_transfer_atdrop) = (elit_On));
            b3 := b3 AND ((state0.dvar_M_sup_S_vacuum) = (elit_Off));
            b2 := b3;
            IF NOT(b2) THEN
                b3 := (state0.dvar_M_sup_A_transfer2droppos) = (elit_Off);
                b3 := b3 AND ((state0.dvar_M_sup_S_Hinitialized) = (elit_On));
                b3 := b3 AND ((state0.dvar_M_sup_S_transfer_athalfway) = (elit_On));
                b3 := b3 AND ((state0.dvar_M_sup_S_transfer_atdrop) = (elit_Off));
                b3 := b3 AND ((state0.dvar_M_sup_S_product4) = (elit_On));
                b3 := b3 AND ((state0.dvar_M_sup_S_xpos_at3) = (elit_On));
                b3 := b3 AND ((state0.dvar_M_sup_S_vacuum) = (elit_Off));
                b2 := b2 OR (b3);
            END_IF;
            IF NOT(b2) THEN
                b3 := (state0.dvar_M_sup_A_transfer2droppos) = (elit_Off);
                b3 := b3 AND ((state0.dvar_M_sup_S_Hinitialized) = (elit_On));
                b3 := b3 AND ((state0.dvar_M_sup_S_transfer_athalfway) = (elit_Off));
                b3 := b3 AND ((state0.dvar_M_sup_S_transfer_atdrop) = (elit_On));
                b3 := b3 AND ((state0.dvar_M_sup_S_vacuum) = (elit_Off));
                b2 := b2 OR (b3);
            END_IF;
            b1 := b1 AND (b2);
        END_IF;
        IF b1 THEN
            progress := TRUE;
            state1 := state0;

            state1.dvar_M_sup_A_transfer2pickpos := elit_On;

            state0 := state1;
        END_IF;
    END_IF;

    // Event "A_turntable_c_off".
    IF NOT progress THEN
        b1 := (state0.dvar_M_sup_A_turntable) = (elit_On);
        b1 := b1 AND ((state0.dvar_M_sup_sup) = (elit_X));
        b1 := b1 AND ((state0.dvar_M_sup_S_Pinitialized) = (elit_On));
        b1 := b1 AND ((state0.dvar_M_sup_S_turntable) = (elit_Off));
        IF b1 THEN
            progress := TRUE;
            state1 := state0;

            state1.dvar_M_sup_A_turntable := elit_Off;

            state0 := state1;
        END_IF;
    END_IF;

    // Event "A_turntable_c_on".
    IF NOT progress THEN
        b1 := (state0.dvar_M_sup_A_turntable) = (elit_Off);
        IF b1 THEN
            b2 := (state0.dvar_M_sup_ClampDrill) = (elit_one2);
            b2 := b2 OR ((state0.dvar_M_sup_ClampDrill) = (elit_nine));
            b1 := b1 AND (b2);
        END_IF;
        b1 := b1 AND ((state0.dvar_M_sup_sup) = (elit_X));
        b1 := b1 AND ((state0.dvar_M_sup_A_eject) = (elit_Off));
        b1 := b1 AND ((state0.dvar_M_sup_S_atinput) = (elit_On));
        b1 := b1 AND ((state0.dvar_M_sup_S_clamp) = (elit_Off));
        b1 := b1 AND ((state0.dvar_M_sup_S_drill_up) = (elit_On));
        b1 := b1 AND ((state0.dvar_M_sup_S_Pinitialized) = (elit_On));
        b1 := b1 AND ((state0.dvar_M_sup_S_turntable) = (elit_On));
        b1 := b1 AND ((state0.dvar_M_sup_Timer) = (elit_Timeout));
        IF b1 THEN
            b2 := (state0.dvar_M_sup_Tester) = (elit_One);
            b2 := b2 OR ((state0.dvar_M_sup_Tester) = (elit_Three));
            b1 := b1 AND (b2);
        END_IF;
        IF b1 THEN
            progress := TRUE;
            state1 := state0;

            state1.dvar_M_sup_A_turntable := elit_On;
            IF ((state0.dvar_M_sup_ClampDrill) = (elit_one2)) THEN
                state1.dvar_M_sup_ClampDrill := elit_one2;
            ELSIF ((state0.dvar_M_sup_ClampDrill) = (elit_nine)) THEN
                state1.dvar_M_sup_ClampDrill := elit_one2;
            END_IF;
            IF ((state0.dvar_M_sup_Tester) = (elit_One)) THEN
                state1.dvar_M_sup_Tester := elit_One;
            ELSIF ((state0.dvar_M_sup_Tester) = (elit_Three)) THEN
                state1.dvar_M_sup_Tester := elit_One;
            END_IF;

            state0 := state1;
        END_IF;
    END_IF;

    // Event "A_vacuum_c_off".
    IF NOT progress THEN
        b1 := (state0.dvar_M_sup_A_vacuum) = (elit_On);
        b1 := b1 AND ((state0.dvar_M_sup_sup) = (elit_X));
        b1 := b1 AND ((state0.dvar_M_sup_S_Hinitialized) = (elit_On));
        b1 := b1 AND ((state0.dvar_M_sup_S_transfer_atdrop) = (elit_On));
        IF b1 THEN
            progress := TRUE;
            state1 := state0;

            state1.dvar_M_sup_A_vacuum := elit_Off;

            state0 := state1;
        END_IF;
    END_IF;

    // Event "A_vacuum_c_on".
    IF NOT progress THEN
        b1 := (state0.dvar_M_sup_A_vacuum) = (elit_Off);
        b1 := b1 AND ((state0.dvar_M_sup_sup) = (elit_X));
        b1 := b1 AND ((state0.dvar_M_sup_S_Hinitialized) = (elit_On));
        b1 := b1 AND ((state0.dvar_M_sup_S_transfer_atpickup) = (elit_On));
        IF b1 THEN
            progress := TRUE;
            state1 := state0;

            state1.dvar_M_sup_A_vacuum := elit_On;

            state0 := state1;
        END_IF;
    END_IF;

    // Event "A_x2distributing_c_off".
    IF NOT progress THEN
        b1 := (state0.dvar_M_sup_A_x2distributing) = (elit_On);
        b1 := b1 AND ((state0.dvar_M_sup_sup) = (elit_X));
        IF b1 THEN
            b3 := (state0.dvar_M_sup_A_x2testing) = (elit_On);
            b3 := b3 AND ((state0.dvar_M_sup_S_Hinitialized) = (elit_On));
            b3 := b3 AND ((state0.dvar_M_sup_S_transfer_athalfway) = (elit_On));
            b3 := b3 AND ((state0.dvar_M_sup_S_product4) = (elit_On));
            b3 := b3 AND ((state0.dvar_M_sup_S_gripper) = (elit_On));
            b3 := b3 AND ((state0.dvar_M_sup_S_xpos_at2) = (elit_On));
            b3 := b3 AND ((state0.dvar_M_sup_S_zpos_atup) = (elit_On));
            b2 := b3;
            IF NOT(b2) THEN
                b3 := (state0.dvar_M_sup_A_x2testing) = (elit_On);
                b3 := b3 AND ((state0.dvar_M_sup_S_Hinitialized) = (elit_On));
                b3 := b3 AND ((state0.dvar_M_sup_S_transfer_athalfway) = (elit_On));
                b3 := b3 AND ((state0.dvar_M_sup_S_product4) = (elit_On));
                b3 := b3 AND ((state0.dvar_M_sup_S_gripper) = (elit_On));
                b3 := b3 AND ((state0.dvar_M_sup_S_xpos_at2) = (elit_Off));
                b3 := b3 AND ((state0.dvar_M_sup_S_xpos_at1) = (elit_On));
                b3 := b3 AND ((state0.dvar_M_sup_S_zpos_atup) = (elit_On));
                b2 := b2 OR (b3);
            END_IF;
            IF NOT(b2) THEN
                b3 := (state0.dvar_M_sup_A_x2testing) = (elit_On);
                b3 := b3 AND ((state0.dvar_M_sup_S_Hinitialized) = (elit_On));
                b3 := b3 AND ((state0.dvar_M_sup_S_transfer_athalfway) = (elit_On));
                b3 := b3 AND ((state0.dvar_M_sup_S_product4) = (elit_Off));
                b3 := b3 AND ((state0.dvar_M_sup_S_gripper) = (elit_On));
                b3 := b3 AND ((state0.dvar_M_sup_S_xpos_at3) = (elit_On));
                b3 := b3 AND ((state0.dvar_M_sup_S_zpos_atup) = (elit_On));
                b2 := b2 OR (b3);
            END_IF;
            IF NOT(b2) THEN
                b3 := (state0.dvar_M_sup_A_x2testing) = (elit_On);
                b3 := b3 AND ((state0.dvar_M_sup_S_Hinitialized) = (elit_On));
                b3 := b3 AND ((state0.dvar_M_sup_S_transfer_athalfway) = (elit_On));
                b3 := b3 AND ((state0.dvar_M_sup_S_product4) = (elit_Off));
                b3 := b3 AND ((state0.dvar_M_sup_S_gripper) = (elit_On));
                b3 := b3 AND ((state0.dvar_M_sup_S_xpos_at3) = (elit_Off));
                b3 := b3 AND ((state0.dvar_M_sup_S_xpos_at2) = (elit_On));
                b3 := b3 AND ((state0.dvar_M_sup_S_zpos_atup) = (elit_On));
                b2 := b2 OR (b3);
            END_IF;
            IF NOT(b2) THEN
                b3 := (state0.dvar_M_sup_A_x2testing) = (elit_On);
                b3 := b3 AND ((state0.dvar_M_sup_S_Hinitialized) = (elit_On));
                b3 := b3 AND ((state0.dvar_M_sup_S_transfer_athalfway) = (elit_On));
                b3 := b3 AND ((state0.dvar_M_sup_S_product4) = (elit_Off));
                b3 := b3 AND ((state0.dvar_M_sup_S_gripper) = (elit_On));
                b3 := b3 AND ((state0.dvar_M_sup_S_xpos_at3) = (elit_Off));
                b3 := b3 AND ((state0.dvar_M_sup_S_xpos_at2) = (elit_Off));
                b3 := b3 AND ((state0.dvar_M_sup_S_xpos_at1) = (elit_On));
                b3 := b3 AND ((state0.dvar_M_sup_S_zpos_atup) = (elit_On));
                b2 := b2 OR (b3);
            END_IF;
            IF NOT(b2) THEN
                b3 := (state0.dvar_M_sup_A_x2testing) = (elit_On);
                b3 := b3 AND ((state0.dvar_M_sup_S_Hinitialized) = (elit_On));
                b3 := b3 AND ((state0.dvar_M_sup_S_transfer_athalfway) = (elit_Off));
                b3 := b3 AND ((state0.dvar_M_sup_S_gripper) = (elit_On));
                b3 := b3 AND ((state0.dvar_M_sup_S_xpos_at2) = (elit_On));
                b3 := b3 AND ((state0.dvar_M_sup_S_zpos_atup) = (elit_On));
                b2 := b2 OR (b3);
            END_IF;
            IF NOT(b2) THEN
                b3 := (state0.dvar_M_sup_A_x2testing) = (elit_On);
                b3 := b3 AND ((state0.dvar_M_sup_S_Hinitialized) = (elit_On));
                b3 := b3 AND ((state0.dvar_M_sup_S_transfer_athalfway) = (elit_Off));
                b3 := b3 AND ((state0.dvar_M_sup_S_gripper) = (elit_On));
                b3 := b3 AND ((state0.dvar_M_sup_S_xpos_at2) = (elit_Off));
                b3 := b3 AND ((state0.dvar_M_sup_S_xpos_at1) = (elit_On));
                b3 := b3 AND ((state0.dvar_M_sup_S_zpos_atup) = (elit_On));
                b2 := b2 OR (b3);
            END_IF;
            b1 := b1 AND (b2);
        END_IF;
        IF b1 THEN
            progress := TRUE;
            state1 := state0;

            state1.dvar_M_sup_A_x2distributing := elit_Off;

            state0 := state1;
        END_IF;
    END_IF;

    // Event "A_x2distributing_c_on".
    IF NOT progress THEN
        b1 := (state0.dvar_M_sup_A_x2distributing) = (elit_Off);
        b1 := b1 AND ((state0.dvar_M_sup_sup) = (elit_X));
        IF b1 THEN
            b2 := (state0.dvar_M_sup_S_Hinitialized) = (elit_Off);
            b2 := b2 OR ((state0.dvar_M_sup_S_transfer_athalfway) = (elit_Off));
            b2 := b2 OR ((state0.dvar_M_sup_S_product4) = (elit_Off));
            b2 := b2 OR ((state0.dvar_M_sup_S_xpos_at3) = (elit_On));
            b2 := b2 OR ((state0.dvar_M_sup_S_xpos_atdrop) = (elit_On));
            b1 := b1 AND (b2);
        END_IF;
        IF b1 THEN
            b2 := (state0.dvar_M_sup_S_Hinitialized) = (elit_Off);
            b2 := b2 OR ((state0.dvar_M_sup_S_transfer_athalfway) = (elit_Off));
            b2 := b2 OR ((state0.dvar_M_sup_S_product4) = (elit_On));
            b2 := b2 OR ((state0.dvar_M_sup_S_xpos_atdrop) = (elit_On));
            b1 := b1 AND (b2);
        END_IF;
        IF b1 THEN
            b2 := (state0.dvar_M_sup_S_Hinitialized) = (elit_Off);
            b2 := b2 OR ((state0.dvar_M_sup_S_transfer_athalfway) = (elit_On));
            b2 := b2 OR ((state0.dvar_M_sup_S_xpos_at3) = (elit_On));
            b2 := b2 OR ((state0.dvar_M_sup_S_xpos_atdrop) = (elit_On));
            b1 := b1 AND (b2);
        END_IF;
        b1 := b1 AND ((state0.dvar_M_sup_S_Hinitialized) = (elit_On));
        IF b1 THEN
            progress := TRUE;
            state1 := state0;

            state1.dvar_M_sup_A_x2distributing := elit_On;

            state0 := state1;
        END_IF;
    END_IF;

    // Event "A_x2testing_c_off".
    IF NOT progress THEN
        b1 := (state0.dvar_M_sup_A_x2testing) = (elit_On);
        b1 := b1 AND ((state0.dvar_M_sup_sup) = (elit_X));
        IF b1 THEN
            b3 := (state0.dvar_M_sup_A_x2distributing) = (elit_On);
            b3 := b3 AND ((state0.dvar_M_sup_S_Hinitialized) = (elit_On));
            b3 := b3 AND ((state0.dvar_M_sup_S_product1) = (elit_On));
            b3 := b3 AND ((state0.dvar_M_sup_S_product2) = (elit_On));
            b3 := b3 AND ((state0.dvar_M_sup_S_product3) = (elit_On));
            b3 := b3 AND ((state0.dvar_M_sup_S_gripper) = (elit_Off));
            b3 := b3 AND ((state0.dvar_M_sup_S_xpos_atdrop) = (elit_On));
            b3 := b3 AND ((state0.dvar_M_sup_S_zpos_atup) = (elit_On));
            b2 := b3;
            IF NOT(b2) THEN
                b3 := (state0.dvar_M_sup_A_x2distributing) = (elit_On);
                b3 := b3 AND ((state0.dvar_M_sup_S_Hinitialized) = (elit_On));
                b3 := b3 AND ((state0.dvar_M_sup_S_product1) = (elit_On));
                b3 := b3 AND ((state0.dvar_M_sup_S_product2) = (elit_On));
                b3 := b3 AND ((state0.dvar_M_sup_S_product3) = (elit_Off));
                b3 := b3 AND ((state0.dvar_M_sup_S_gripper) = (elit_Off));
                b3 := b3 AND ((state0.dvar_M_sup_S_xpos_at3) = (elit_On));
                b3 := b3 AND ((state0.dvar_M_sup_S_zpos_atup) = (elit_On));
                b2 := b2 OR (b3);
            END_IF;
            IF NOT(b2) THEN
                b3 := (state0.dvar_M_sup_A_x2distributing) = (elit_On);
                b3 := b3 AND ((state0.dvar_M_sup_S_Hinitialized) = (elit_On));
                b3 := b3 AND ((state0.dvar_M_sup_S_product1) = (elit_On));
                b3 := b3 AND ((state0.dvar_M_sup_S_product2) = (elit_On));
                b3 := b3 AND ((state0.dvar_M_sup_S_product3) = (elit_Off));
                b3 := b3 AND ((state0.dvar_M_sup_S_gripper) = (elit_Off));
                b3 := b3 AND ((state0.dvar_M_sup_S_xpos_at3) = (elit_Off));
                b3 := b3 AND ((state0.dvar_M_sup_S_xpos_atdrop) = (elit_On));
                b3 := b3 AND ((state0.dvar_M_sup_S_zpos_atup) = (elit_On));
                b2 := b2 OR (b3);
            END_IF;
            IF NOT(b2) THEN
                b3 := (state0.dvar_M_sup_A_x2distributing) = (elit_On);
                b3 := b3 AND ((state0.dvar_M_sup_S_Hinitialized) = (elit_On));
                b3 := b3 AND ((state0.dvar_M_sup_S_product1) = (elit_On));
                b3 := b3 AND ((state0.dvar_M_sup_S_product2) = (elit_Off));
                b3 := b3 AND ((state0.dvar_M_sup_S_product3) = (elit_On));
                b3 := b3 AND ((state0.dvar_M_sup_S_gripper) = (elit_Off));
                b3 := b3 AND ((state0.dvar_M_sup_S_xpos_at2) = (elit_On));
                b3 := b3 AND ((state0.dvar_M_sup_S_zpos_atup) = (elit_On));
                b2 := b2 OR (b3);
            END_IF;
            IF NOT(b2) THEN
                b3 := (state0.dvar_M_sup_A_x2distributing) = (elit_On);
                b3 := b3 AND ((state0.dvar_M_sup_S_Hinitialized) = (elit_On));
                b3 := b3 AND ((state0.dvar_M_sup_S_product1) = (elit_On));
                b3 := b3 AND ((state0.dvar_M_sup_S_product2) = (elit_Off));
                b3 := b3 AND ((state0.dvar_M_sup_S_product3) = (elit_On));
                b3 := b3 AND ((state0.dvar_M_sup_S_gripper) = (elit_Off));
                b3 := b3 AND ((state0.dvar_M_sup_S_xpos_at2) = (elit_Off));
                b3 := b3 AND ((state0.dvar_M_sup_S_xpos_atdrop) = (elit_On));
                b3 := b3 AND ((state0.dvar_M_sup_S_zpos_atup) = (elit_On));
                b2 := b2 OR (b3);
            END_IF;
            IF NOT(b2) THEN
                b3 := (state0.dvar_M_sup_A_x2distributing) = (elit_On);
                b3 := b3 AND ((state0.dvar_M_sup_S_Hinitialized) = (elit_On));
                b3 := b3 AND ((state0.dvar_M_sup_S_product1) = (elit_On));
                b3 := b3 AND ((state0.dvar_M_sup_S_product2) = (elit_Off));
                b3 := b3 AND ((state0.dvar_M_sup_S_product3) = (elit_Off));
                b3 := b3 AND ((state0.dvar_M_sup_S_gripper) = (elit_Off));
                b3 := b3 AND ((state0.dvar_M_sup_S_xpos_at3) = (elit_On));
                b3 := b3 AND ((state0.dvar_M_sup_S_zpos_atup) = (elit_On));
                b2 := b2 OR (b3);
            END_IF;
            IF NOT(b2) THEN
                b3 := (state0.dvar_M_sup_A_x2distributing) = (elit_On);
                b3 := b3 AND ((state0.dvar_M_sup_S_Hinitialized) = (elit_On));
                b3 := b3 AND ((state0.dvar_M_sup_S_product1) = (elit_On));
                b3 := b3 AND ((state0.dvar_M_sup_S_product2) = (elit_Off));
                b3 := b3 AND ((state0.dvar_M_sup_S_product3) = (elit_Off));
                b3 := b3 AND ((state0.dvar_M_sup_S_gripper) = (elit_Off));
                b3 := b3 AND ((state0.dvar_M_sup_S_xpos_at3) = (elit_Off));
                b3 := b3 AND ((state0.dvar_M_sup_S_xpos_at2) = (elit_On));
                b3 := b3 AND ((state0.dvar_M_sup_S_zpos_atup) = (elit_On));
                b2 := b2 OR (b3);
            END_IF;
            IF NOT(b2) THEN
                b3 := (state0.dvar_M_sup_A_x2distributing) = (elit_On);
                b3 := b3 AND ((state0.dvar_M_sup_S_Hinitialized) = (elit_On));
                b3 := b3 AND ((state0.dvar_M_sup_S_product1) = (elit_On));
                b3 := b3 AND ((state0.dvar_M_sup_S_product2) = (elit_Off));
                b3 := b3 AND ((state0.dvar_M_sup_S_product3) = (elit_Off));
                b3 := b3 AND ((state0.dvar_M_sup_S_gripper) = (elit_Off));
                b3 := b3 AND ((state0.dvar_M_sup_S_xpos_at3) = (elit_Off));
                b3 := b3 AND ((state0.dvar_M_sup_S_xpos_at2) = (elit_Off));
                b3 := b3 AND ((state0.dvar_M_sup_S_xpos_atdrop) = (elit_On));
                b3 := b3 AND ((state0.dvar_M_sup_S_zpos_atup) = (elit_On));
                b2 := b2 OR (b3);
            END_IF;
            IF NOT(b2) THEN
                b3 := (state0.dvar_M_sup_A_x2distributing) = (elit_On);
                b3 := b3 AND ((state0.dvar_M_sup_S_Hinitialized) = (elit_On));
                b3 := b3 AND ((state0.dvar_M_sup_S_product1) = (elit_Off));
                b3 := b3 AND ((state0.dvar_M_sup_S_product2) = (elit_On));
                b3 := b3 AND ((state0.dvar_M_sup_S_product3) = (elit_On));
                b3 := b3 AND ((state0.dvar_M_sup_S_gripper) = (elit_Off));
                b3 := b3 AND ((state0.dvar_M_sup_S_xpos_atdrop) = (elit_On));
                b3 := b3 AND ((state0.dvar_M_sup_S_zpos_atup) = (elit_On));
                b2 := b2 OR (b3);
            END_IF;
            IF NOT(b2) THEN
                b3 := (state0.dvar_M_sup_A_x2distributing) = (elit_On);
                b3 := b3 AND ((state0.dvar_M_sup_S_Hinitialized) = (elit_On));
                b3 := b3 AND ((state0.dvar_M_sup_S_product1) = (elit_Off));
                b3 := b3 AND ((state0.dvar_M_sup_S_product2) = (elit_On));
                b3 := b3 AND ((state0.dvar_M_sup_S_product3) = (elit_Off));
                b3 := b3 AND ((state0.dvar_M_sup_S_gripper) = (elit_Off));
                b3 := b3 AND ((state0.dvar_M_sup_S_xpos_at3) = (elit_On));
                b3 := b3 AND ((state0.dvar_M_sup_S_zpos_atup) = (elit_On));
                b2 := b2 OR (b3);
            END_IF;
            IF NOT(b2) THEN
                b3 := (state0.dvar_M_sup_A_x2distributing) = (elit_On);
                b3 := b3 AND ((state0.dvar_M_sup_S_Hinitialized) = (elit_On));
                b3 := b3 AND ((state0.dvar_M_sup_S_product1) = (elit_Off));
                b3 := b3 AND ((state0.dvar_M_sup_S_product2) = (elit_On));
                b3 := b3 AND ((state0.dvar_M_sup_S_product3) = (elit_Off));
                b3 := b3 AND ((state0.dvar_M_sup_S_gripper) = (elit_Off));
                b3 := b3 AND ((state0.dvar_M_sup_S_xpos_at3) = (elit_Off));
                b3 := b3 AND ((state0.dvar_M_sup_S_xpos_atdrop) = (elit_On));
                b3 := b3 AND ((state0.dvar_M_sup_S_zpos_atup) = (elit_On));
                b2 := b2 OR (b3);
            END_IF;
            IF NOT(b2) THEN
                b3 := (state0.dvar_M_sup_A_x2distributing) = (elit_On);
                b3 := b3 AND ((state0.dvar_M_sup_S_Hinitialized) = (elit_On));
                b3 := b3 AND ((state0.dvar_M_sup_S_product1) = (elit_Off));
                b3 := b3 AND ((state0.dvar_M_sup_S_product2) = (elit_Off));
                b3 := b3 AND ((state0.dvar_M_sup_S_gripper) = (elit_Off));
                b3 := b3 AND ((state0.dvar_M_sup_S_xpos_atdrop) = (elit_On));
                b3 := b3 AND ((state0.dvar_M_sup_S_zpos_atup) = (elit_On));
                b2 := b2 OR (b3);
            END_IF;
            b1 := b1 AND (b2);
        END_IF;
        IF b1 THEN
            progress := TRUE;
            state1 := state0;

            state1.dvar_M_sup_A_x2testing := elit_Off;

            state0 := state1;
        END_IF;
    END_IF;

    // Event "A_x2testing_c_on".
    IF NOT progress THEN
        b1 := (state0.dvar_M_sup_A_x2testing) = (elit_Off);
        b1 := b1 AND ((state0.dvar_M_sup_sup) = (elit_X));
        IF b1 THEN
            b2 := (state0.dvar_M_sup_S_Hinitialized) = (elit_Off);
            b2 := b2 OR ((state0.dvar_M_sup_S_product1) = (elit_Off));
            b2 := b2 OR ((state0.dvar_M_sup_S_product2) = (elit_Off));
            b2 := b2 OR ((state0.dvar_M_sup_S_product3) = (elit_Off));
            b2 := b2 OR ((state0.dvar_M_sup_S_xpos_at3) = (elit_On));
            b2 := b2 OR ((state0.dvar_M_sup_S_xpos_at2) = (elit_On));
            b2 := b2 OR ((state0.dvar_M_sup_S_xpos_at1) = (elit_On));
            b1 := b1 AND (b2);
        END_IF;
        IF b1 THEN
            b2 := (state0.dvar_M_sup_S_Hinitialized) = (elit_Off);
            b2 := b2 OR ((state0.dvar_M_sup_S_product1) = (elit_Off));
            b2 := b2 OR ((state0.dvar_M_sup_S_product2) = (elit_Off));
            b2 := b2 OR ((state0.dvar_M_sup_S_product3) = (elit_On));
            b2 := b2 OR ((state0.dvar_M_sup_S_xpos_at2) = (elit_On));
            b2 := b2 OR ((state0.dvar_M_sup_S_xpos_at1) = (elit_On));
            b1 := b1 AND (b2);
        END_IF;
        IF b1 THEN
            b2 := (state0.dvar_M_sup_S_Hinitialized) = (elit_Off);
            b2 := b2 OR ((state0.dvar_M_sup_S_product1) = (elit_Off));
            b2 := b2 OR ((state0.dvar_M_sup_S_product2) = (elit_On));
            b2 := b2 OR ((state0.dvar_M_sup_S_product3) = (elit_Off));
            b2 := b2 OR ((state0.dvar_M_sup_S_xpos_at3) = (elit_On));
            b2 := b2 OR ((state0.dvar_M_sup_S_xpos_at1) = (elit_On));
            b1 := b1 AND (b2);
        END_IF;
        IF b1 THEN
            b2 := (state0.dvar_M_sup_S_Hinitialized) = (elit_Off);
            b2 := b2 OR ((state0.dvar_M_sup_S_product1) = (elit_Off));
            b2 := b2 OR ((state0.dvar_M_sup_S_product2) = (elit_On));
            b2 := b2 OR ((state0.dvar_M_sup_S_product3) = (elit_On));
            b2 := b2 OR ((state0.dvar_M_sup_S_xpos_at1) = (elit_On));
            b1 := b1 AND (b2);
        END_IF;
        IF b1 THEN
            b2 := (state0.dvar_M_sup_S_Hinitialized) = (elit_Off);
            b2 := b2 OR ((state0.dvar_M_sup_S_product1) = (elit_On));
            b2 := b2 OR ((state0.dvar_M_sup_S_product2) = (elit_Off));
            b2 := b2 OR ((state0.dvar_M_sup_S_product3) = (elit_Off));
            b2 := b2 OR ((state0.dvar_M_sup_S_xpos_at3) = (elit_On));
            b2 := b2 OR ((state0.dvar_M_sup_S_xpos_at2) = (elit_On));
            b2 := b2 OR ((state0.dvar_M_sup_S_xpos_at1) = (elit_On));
            b1 := b1 AND (b2);
        END_IF;
        IF b1 THEN
            b2 := (state0.dvar_M_sup_S_Hinitialized) = (elit_Off);
            b2 := b2 OR ((state0.dvar_M_sup_S_product1) = (elit_On));
            b2 := b2 OR ((state0.dvar_M_sup_S_product2) = (elit_Off));
            b2 := b2 OR ((state0.dvar_M_sup_S_product3) = (elit_On));
            b2 := b2 OR ((state0.dvar_M_sup_S_xpos_at2) = (elit_On));
            b2 := b2 OR ((state0.dvar_M_sup_S_xpos_at1) = (elit_On));
            b1 := b1 AND (b2);
        END_IF;
        IF b1 THEN
            b2 := (state0.dvar_M_sup_S_Hinitialized) = (elit_Off);
            b2 := b2 OR ((state0.dvar_M_sup_S_product1) = (elit_On));
            b2 := b2 OR ((state0.dvar_M_sup_S_product2) = (elit_On));
            b2 := b2 OR ((state0.dvar_M_sup_S_xpos_at3) = (elit_On));
            b2 := b2 OR ((state0.dvar_M_sup_S_xpos_at1) = (elit_On));
            b1 := b1 AND (b2);
        END_IF;
        b1 := b1 AND ((state0.dvar_M_sup_S_Hinitialized) = (elit_On));
        IF b1 THEN
            progress := TRUE;
            state1 := state0;

            state1.dvar_M_sup_A_x2testing := elit_On;

            state0 := state1;
        END_IF;
    END_IF;

    // Event "A_zdown_c_off".
    IF NOT progress THEN
        b1 := (state0.dvar_M_sup_A_zdown) = (elit_On);
        b1 := b1 AND ((state0.dvar_M_sup_sup) = (elit_X));
        IF b1 THEN
            b3 := (state0.dvar_M_sup_S_Hinitialized) = (elit_On);
            b3 := b3 AND ((state0.dvar_M_sup_A_gripperclose) = (elit_On));
            b3 := b3 AND ((state0.dvar_M_sup_S_gripper) = (elit_On));
            b3 := b3 AND ((state0.dvar_M_sup_S_xpos_at3) = (elit_On));
            b3 := b3 AND ((state0.dvar_M_sup_S_zpos_atdown) = (elit_On));
            b2 := b3;
            IF NOT(b2) THEN
                b3 := (state0.dvar_M_sup_S_Hinitialized) = (elit_On);
                b3 := b3 AND ((state0.dvar_M_sup_A_gripperclose) = (elit_On));
                b3 := b3 AND ((state0.dvar_M_sup_S_gripper) = (elit_On));
                b3 := b3 AND ((state0.dvar_M_sup_S_xpos_at3) = (elit_Off));
                b3 := b3 AND ((state0.dvar_M_sup_S_xpos_at2) = (elit_On));
                b3 := b3 AND ((state0.dvar_M_sup_S_zpos_atdown) = (elit_On));
                b2 := b2 OR (b3);
            END_IF;
            IF NOT(b2) THEN
                b3 := (state0.dvar_M_sup_S_Hinitialized) = (elit_On);
                b3 := b3 AND ((state0.dvar_M_sup_A_gripperclose) = (elit_On));
                b3 := b3 AND ((state0.dvar_M_sup_S_gripper) = (elit_On));
                b3 := b3 AND ((state0.dvar_M_sup_S_xpos_at3) = (elit_Off));
                b3 := b3 AND ((state0.dvar_M_sup_S_xpos_at2) = (elit_Off));
                b3 := b3 AND ((state0.dvar_M_sup_S_xpos_at1) = (elit_On));
                b3 := b3 AND ((state0.dvar_M_sup_S_zpos_atdown) = (elit_On));
                b2 := b2 OR (b3);
            END_IF;
            IF NOT(b2) THEN
                b3 := (state0.dvar_M_sup_S_Hinitialized) = (elit_On);
                b3 := b3 AND ((state0.dvar_M_sup_A_gripperclose) = (elit_Off));
                b3 := b3 AND ((state0.dvar_M_sup_S_xpos_atdrop) = (elit_On));
                b3 := b3 AND ((state0.dvar_M_sup_S_zpos_atdown) = (elit_On));
                b2 := b2 OR (b3);
            END_IF;
            b1 := b1 AND (b2);
        END_IF;
        IF b1 THEN
            progress := TRUE;
            state1 := state0;

            state1.dvar_M_sup_A_zdown := elit_Off;

            state0 := state1;
        END_IF;
    END_IF;

